Yaskawa INFORM job: A_ROOF_SIDE_0617_2_PAINT_4.JBI

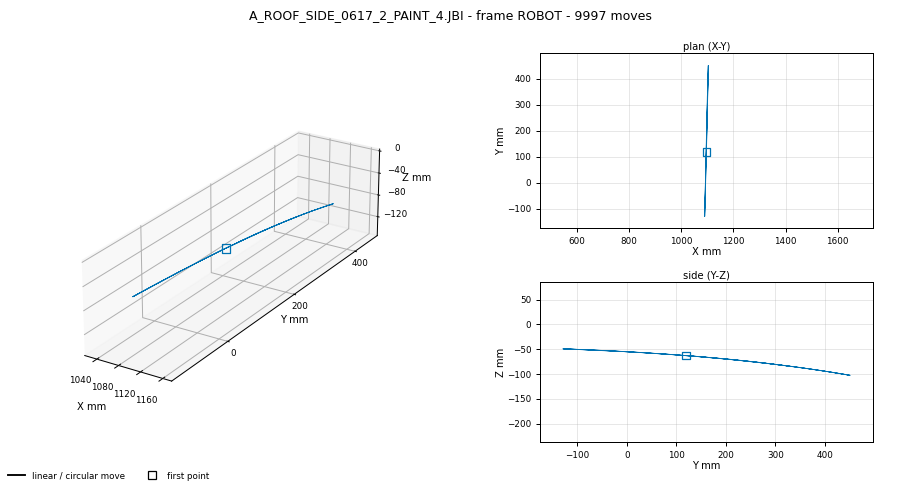
[picture p0: tool path of A_ROOF_SIDE_0617_2_PAINT_4.JBI in frame ROBOT, 9997 of 9997 moves have a stored position in this frame; points joined in program order, loops and branches not executed]
/JOB
//NAME A_ROOF_SIDE_0617_2_PAINT4
//POS
///NPOS 9997,0,0,0,0,0
///TOOL 1
///USER 0
///POSTYPE ROBOT
///RECTAN
///RCONF 1,0,0,0,0,0,0,0,0,0,0,0,0,0,0,0,0,0,0,0,0,0,0,0
C00000=1096.591,119.908,-62.578,176.519,16.757,152.269
C00001=1096.596,120.158,-62.598,176.522,16.758,152.268
C00002=1096.602,120.407,-62.618,176.524,16.758,152.268
C00003=1096.608,120.656,-62.637,176.527,16.758,152.267
C00004=1096.614,120.905,-62.656,176.530,16.759,152.267
C00005=1096.619,121.154,-62.675,176.533,16.759,152.267
C00006=1096.625,121.404,-62.694,176.536,16.760,152.266
C00007=1096.630,121.653,-62.713,176.539,16.761,152.266
C00008=1096.636,121.902,-62.733,176.541,16.761,152.265
C00009=1096.641,122.152,-62.753,176.544,16.762,152.265
C00010=1096.646,122.400,-62.772,176.546,16.761,152.264
C00011=1096.652,122.650,-62.791,176.549,16.762,152.264
C00012=1096.658,122.899,-62.811,176.552,16.763,152.263
C00013=1096.664,123.148,-62.830,176.555,16.763,152.263
C00014=1096.669,123.397,-62.850,176.558,16.764,152.262
C00015=1096.675,123.647,-62.869,176.561,16.764,152.262
C00016=1096.681,123.896,-62.889,176.563,16.765,152.262
C00017=1096.686,124.144,-62.908,176.566,16.765,152.261
C00018=1096.692,124.394,-62.927,176.569,16.766,152.261
C00019=1096.697,124.643,-62.946,176.571,16.766,152.260
C00020=1096.703,124.892,-62.966,176.575,16.766,152.260
C00021=1096.709,125.141,-62.985,176.578,16.767,152.259
C00022=1096.715,125.391,-63.005,176.580,16.767,152.259
C00023=1096.720,125.640,-63.025,176.583,16.768,152.258
C00024=1096.726,125.889,-63.045,176.585,16.768,152.258
C00025=1096.731,126.138,-63.064,176.589,16.768,152.257
C00026=1096.737,126.387,-63.083,176.592,16.769,152.257
C00027=1096.743,126.636,-63.103,176.594,16.769,152.256
C00028=1096.749,126.885,-63.123,176.597,16.770,152.256
C00029=1096.754,127.135,-63.142,176.600,16.770,152.256
C00030=1096.760,127.383,-63.162,176.602,16.770,152.255
C00031=1096.766,127.659,-63.183,176.606,16.771,152.254
C00032=1096.773,127.934,-63.205,176.609,16.771,152.254
C00033=1096.779,128.209,-63.226,176.612,16.772,152.253
C00034=1096.785,128.484,-63.249,176.615,16.772,152.253
C00035=1096.791,128.733,-63.269,176.618,16.773,152.252
C00036=1096.796,128.982,-63.288,176.621,16.773,152.252
C00037=1096.802,129.231,-63.307,176.624,16.773,152.251
C00038=1096.808,129.480,-63.327,176.627,16.774,152.251
C00039=1096.814,129.729,-63.347,176.629,16.774,152.250
C00040=1096.819,129.979,-63.366,176.632,16.774,152.250
C00041=1096.825,130.227,-63.386,176.636,16.775,152.249
C00042=1096.830,130.477,-63.406,176.638,16.775,152.249
C00043=1096.836,130.726,-63.426,176.641,16.775,152.248
C00044=1096.842,130.975,-63.445,176.644,16.776,152.248
C00045=1096.848,131.225,-63.465,176.646,16.776,152.247
C00046=1096.854,131.474,-63.486,176.649,16.777,152.247
C00047=1096.859,131.723,-63.505,176.653,16.777,152.246
C00048=1096.865,131.972,-63.525,176.655,16.777,152.246
C00049=1096.871,132.221,-63.544,176.658,16.778,152.245
C00050=1096.876,132.470,-63.565,176.661,16.778,152.245
C00051=1096.882,132.719,-63.585,176.664,16.778,152.244
C00052=1096.888,132.969,-63.604,176.667,16.778,152.244
C00053=1096.893,133.218,-63.624,176.670,16.779,152.243
C00054=1096.899,133.467,-63.644,176.672,16.779,152.243
C00055=1096.904,133.716,-63.664,176.676,16.779,152.242
C00056=1096.910,133.965,-63.684,176.679,16.780,152.242
C00057=1096.916,134.214,-63.704,176.681,16.780,152.241
C00058=1096.921,134.464,-63.724,176.684,16.781,152.241
C00059=1096.927,134.713,-63.744,176.687,16.781,152.240
C00060=1096.932,134.962,-63.765,176.690,16.781,152.240
C00061=1096.938,135.211,-63.784,176.693,16.782,152.239
C00062=1096.944,135.460,-63.804,176.696,16.782,152.239
C00063=1096.949,135.709,-63.824,176.698,16.782,152.238
C00064=1096.955,135.958,-63.844,176.701,16.783,152.238
C00065=1096.961,136.207,-63.865,176.705,16.783,152.237
C00066=1096.966,136.456,-63.884,176.707,16.783,152.237
C00067=1096.972,136.706,-63.905,176.710,16.784,152.236
C00068=1096.978,136.954,-63.925,176.713,16.784,152.236
C00069=1096.983,137.204,-63.945,176.716,16.785,152.235
C00070=1096.989,137.452,-63.965,176.719,16.785,152.235
C00071=1096.994,137.702,-63.984,176.722,16.785,152.234
C00072=1097.000,137.951,-64.005,176.725,16.785,152.234
C00073=1097.006,138.200,-64.025,176.727,16.785,152.233
C00074=1097.012,138.450,-64.046,176.731,16.786,152.233
C00075=1097.018,138.698,-64.066,176.734,16.786,152.232
C00076=1097.023,138.947,-64.086,176.736,16.786,152.232
C00077=1097.029,139.196,-64.106,176.739,16.787,152.231
C00078=1097.034,139.446,-64.126,176.743,16.787,152.231
C00079=1097.039,139.695,-64.147,176.745,16.787,152.230
C00080=1097.045,139.944,-64.167,176.748,16.788,152.230
C00081=1097.050,140.193,-64.187,176.751,16.788,152.229
C00082=1097.056,140.442,-64.207,176.755,16.788,152.228
C00083=1097.062,140.692,-64.228,176.757,16.788,152.228
C00084=1097.068,140.941,-64.248,176.760,16.789,152.227
C00085=1097.073,141.190,-64.269,176.763,16.789,152.227
C00086=1097.079,141.439,-64.289,176.766,16.789,152.226
C00087=1097.085,141.688,-64.309,176.769,16.790,152.226
C00088=1097.090,141.937,-64.330,176.772,16.790,152.225
C00089=1097.095,142.186,-64.350,176.775,16.790,152.225
C00090=1097.101,142.435,-64.370,176.778,16.790,152.224
C00091=1097.107,142.684,-64.391,176.781,16.791,152.224
C00092=1097.112,142.934,-64.412,176.784,16.791,152.223
C00093=1097.118,143.182,-64.432,176.786,16.791,152.223
C00094=1097.124,143.432,-64.452,176.790,16.792,152.222
C00095=1097.130,143.707,-64.475,176.793,16.792,152.222
C00096=1097.136,143.981,-64.497,176.797,16.792,152.221
C00097=1097.142,144.256,-64.520,176.800,16.792,152.220
C00098=1097.149,144.530,-64.542,176.803,16.793,152.220
C00099=1097.154,144.780,-64.563,176.806,16.793,152.219
C00100=1097.160,145.029,-64.584,176.809,16.793,152.219
C00101=1097.165,145.278,-64.604,176.812,16.793,152.218
C00102=1097.171,145.527,-64.624,176.815,16.794,152.218
C00103=1097.176,145.776,-64.645,176.817,16.794,152.217
C00104=1097.182,146.025,-64.667,176.821,16.794,152.216
C00105=1097.188,146.274,-64.686,176.824,16.795,152.216
C00106=1097.194,146.523,-64.707,176.827,16.795,152.215
C00107=1097.199,146.772,-64.728,176.830,16.795,152.215
C00108=1097.205,147.022,-64.749,176.833,16.795,152.214
C00109=1097.211,147.270,-64.769,176.836,16.795,152.214
C00110=1097.216,147.519,-64.790,176.839,16.795,152.213
C00111=1097.222,147.769,-64.810,176.842,16.796,152.213
C00112=1097.227,148.018,-64.831,176.845,16.796,152.212
C00113=1097.234,148.267,-64.852,176.848,16.796,152.211
C00114=1097.239,148.516,-64.872,176.851,16.796,152.211
C00115=1097.244,148.765,-64.893,176.854,16.796,152.210
C00116=1097.250,149.015,-64.914,176.857,16.797,152.210
C00117=1097.256,149.263,-64.935,176.861,16.797,152.209
C00118=1097.261,149.512,-64.956,176.863,16.797,152.209
C00119=1097.266,149.761,-64.976,176.866,16.797,152.208
C00120=1097.273,150.010,-64.997,176.870,16.798,152.207
C00121=1097.278,150.259,-65.018,176.872,16.797,152.207
C00122=1097.284,150.509,-65.038,176.875,16.798,152.206
C00123=1097.289,150.757,-65.060,176.879,16.798,152.206
C00124=1097.295,151.007,-65.081,176.882,16.799,152.205
C00125=1097.301,151.255,-65.102,176.884,16.798,152.205
C00126=1097.306,151.505,-65.122,176.888,16.799,152.204
C00127=1097.312,151.754,-65.143,176.891,16.799,152.203
C00128=1097.317,152.003,-65.165,176.894,16.799,152.203
C00129=1097.322,152.252,-65.185,176.897,16.799,152.202
C00130=1097.329,152.501,-65.207,176.900,16.800,152.202
C00131=1097.334,152.750,-65.227,176.903,16.800,152.201
C00132=1097.339,152.999,-65.249,176.906,16.800,152.201
C00133=1097.345,153.248,-65.269,176.909,16.800,152.200
C00134=1097.351,153.497,-65.290,176.912,16.801,152.200
C00135=1097.357,153.746,-65.311,176.915,16.801,152.199
C00136=1097.362,153.995,-65.331,176.918,16.800,152.198
C00137=1097.368,154.244,-65.353,176.921,16.801,152.198
C00138=1097.374,154.493,-65.374,176.925,16.801,152.197
C00139=1097.380,154.743,-65.395,176.928,16.801,152.197
C00140=1097.385,154.991,-65.416,176.930,16.801,152.196
C00141=1097.391,155.240,-65.437,176.934,16.801,152.195
C00142=1097.397,155.489,-65.459,176.937,16.802,152.195
C00143=1097.402,155.739,-65.479,176.940,16.802,152.194
C00144=1097.407,155.987,-65.501,176.943,16.802,152.194
C00145=1097.413,156.237,-65.522,176.946,16.802,152.193
C00146=1097.418,156.486,-65.543,176.949,16.802,152.192
C00147=1097.424,156.735,-65.565,176.953,16.803,152.192
C00148=1097.430,156.984,-65.585,176.955,16.802,152.191
C00149=1097.435,157.233,-65.607,176.958,16.803,152.191
C00150=1097.441,157.482,-65.628,176.962,16.803,152.190
C00151=1097.447,157.731,-65.649,176.965,16.803,152.190
C00152=1097.452,157.979,-65.670,176.968,16.803,152.189
C00153=1097.458,158.229,-65.692,176.971,16.803,152.188
C00154=1097.463,158.478,-65.713,176.974,16.804,152.188
C00155=1097.469,158.727,-65.735,176.978,16.804,152.187
C00156=1097.475,158.976,-65.756,176.980,16.803,152.187
C00157=1097.480,159.226,-65.777,176.983,16.804,152.186
C00158=1097.486,159.474,-65.798,176.987,16.804,152.185
C00159=1097.493,159.748,-65.822,176.990,16.804,152.185
C00160=1097.499,160.023,-65.845,176.994,16.804,152.184
C00161=1097.505,160.298,-65.868,176.997,16.804,152.183
C00162=1097.510,160.572,-65.893,177.001,16.804,152.183
C00163=1097.517,160.822,-65.914,177.004,16.805,152.182
C00164=1097.522,161.070,-65.936,177.007,16.805,152.181
C00165=1097.528,161.320,-65.956,177.010,16.804,152.181
C00166=1097.533,161.568,-65.978,177.013,16.805,152.180
C00167=1097.538,161.817,-66.000,177.016,16.805,152.180
C00168=1097.544,162.066,-66.021,177.020,16.805,152.179
C00169=1097.550,162.315,-66.042,177.023,16.805,152.178
C00170=1097.555,162.564,-66.065,177.026,16.805,152.178
C00171=1097.561,162.814,-66.085,177.029,16.806,152.177
C00172=1097.566,163.063,-66.107,177.032,16.806,152.177
C00173=1097.572,163.312,-66.129,177.036,16.806,152.176
C00174=1097.577,163.560,-66.150,177.038,16.806,152.175
C00175=1097.583,163.810,-66.172,177.041,16.806,152.175
C00176=1097.588,164.058,-66.194,177.045,16.806,152.174
C00177=1097.594,164.308,-66.216,177.048,16.806,152.174
C00178=1097.599,164.556,-66.237,177.051,16.807,152.173
C00179=1097.605,164.806,-66.259,177.054,16.807,152.173
C00180=1097.610,165.054,-66.281,177.057,16.807,152.172
C00181=1097.616,165.303,-66.302,177.061,16.807,152.171
C00182=1097.621,165.552,-66.324,177.064,16.807,152.171
C00183=1097.627,165.801,-66.346,177.067,16.808,152.170
C00184=1097.632,166.050,-66.368,177.070,16.807,152.169
C00185=1097.638,166.299,-66.389,177.073,16.807,152.169
C00186=1097.643,166.548,-66.411,177.076,16.808,152.168
C00187=1097.649,166.797,-66.433,177.080,16.808,152.168
C00188=1097.654,167.046,-66.455,177.083,16.808,152.167
C00189=1097.660,167.295,-66.476,177.086,16.807,152.166
C00190=1097.665,167.544,-66.498,177.089,16.808,152.166
C00191=1097.671,167.793,-66.520,177.093,16.808,152.165
C00192=1097.676,168.042,-66.542,177.096,16.808,152.164
C00193=1097.682,168.291,-66.563,177.099,16.809,152.164
C00194=1097.687,168.540,-66.585,177.102,16.808,152.163
C00195=1097.693,168.790,-66.607,177.105,16.808,152.163
C00196=1097.698,169.038,-66.629,177.109,16.809,152.162
C00197=1097.704,169.288,-66.650,177.112,16.809,152.161
C00198=1097.709,169.536,-66.673,177.115,16.808,152.161
C00199=1097.716,169.785,-66.694,177.118,16.808,152.160
C00200=1097.721,170.034,-66.717,177.121,16.809,152.159
C00201=1097.727,170.283,-66.738,177.125,16.809,152.159
C00202=1097.732,170.532,-66.760,177.128,16.809,152.158
C00203=1097.738,170.780,-66.782,177.131,16.808,152.158
C00204=1097.743,171.030,-66.804,177.134,16.809,152.157
C00205=1097.749,171.279,-66.827,177.138,16.809,152.156
C00206=1097.754,171.528,-66.848,177.141,16.809,152.156
C00207=1097.760,171.777,-66.871,177.144,16.809,152.155
C00208=1097.766,172.026,-66.892,177.148,16.809,152.154
C00209=1097.771,172.275,-66.914,177.150,16.809,152.154
C00210=1097.777,172.524,-66.936,177.154,16.809,152.153
C00211=1097.782,172.772,-66.958,177.157,16.809,152.152
C00212=1097.788,173.022,-66.981,177.161,16.810,152.152
C00213=1097.794,173.271,-67.002,177.164,16.809,152.151
C00214=1097.799,173.519,-67.025,177.167,16.809,152.150
C00215=1097.805,173.768,-67.047,177.170,16.809,152.150
C00216=1097.811,174.018,-67.069,177.174,16.809,152.149
C00217=1097.816,174.267,-67.092,177.177,16.810,152.149
C00218=1097.822,174.515,-67.113,177.180,16.809,152.148
C00219=1097.827,174.765,-67.135,177.183,16.809,152.147
C00220=1097.833,175.014,-67.158,177.186,16.809,152.147
C00221=1097.839,175.262,-67.179,177.190,16.809,152.146
C00222=1097.844,175.511,-67.202,177.193,16.809,152.145
C00223=1097.851,175.785,-67.226,177.197,16.809,152.144
C00224=1097.857,176.060,-67.251,177.201,16.809,152.144
C00225=1097.864,176.334,-67.276,177.204,16.809,152.143
C00226=1097.869,176.608,-67.300,177.208,16.809,152.142
C00227=1097.875,176.857,-67.323,177.211,16.809,152.142
C00228=1097.881,177.106,-67.344,177.214,16.809,152.141
C00229=1097.887,177.355,-67.367,177.218,16.809,152.140
C00230=1097.892,177.604,-67.389,177.222,16.809,152.140
C00231=1097.898,177.852,-67.411,177.224,16.809,152.139
C00232=1097.903,178.102,-67.434,177.228,16.809,152.138
C00233=1097.909,178.351,-67.457,177.231,16.809,152.138
C00234=1097.914,178.600,-67.479,177.234,16.809,152.137
C00235=1097.920,178.848,-67.501,177.238,16.809,152.136
C00236=1097.926,179.097,-67.524,177.241,16.809,152.136
C00237=1097.931,179.346,-67.546,177.244,16.808,152.135
C00238=1097.938,179.595,-67.568,177.248,16.808,152.134
C00239=1097.943,179.845,-67.591,177.251,16.809,152.134
C00240=1097.949,180.093,-67.614,177.254,16.809,152.133
C00241=1097.954,180.342,-67.636,177.258,16.809,152.132
C00242=1097.960,180.591,-67.658,177.262,16.809,152.131
C00243=1097.966,180.840,-67.681,177.264,16.808,152.131
C00244=1097.972,181.089,-67.704,177.268,16.808,152.130
C00245=1097.977,181.338,-67.726,177.271,16.808,152.129
C00246=1097.984,181.587,-67.748,177.275,16.808,152.129
C00247=1097.989,181.836,-67.771,177.278,16.808,152.128
C00248=1097.994,182.084,-67.793,177.282,16.808,152.127
C00249=1098.000,182.333,-67.816,177.284,16.808,152.127
C00250=1098.006,182.582,-67.838,177.288,16.808,152.126
C00251=1098.012,182.831,-67.861,177.291,16.808,152.125
C00252=1098.018,183.080,-67.883,177.295,16.808,152.125
C00253=1098.023,183.329,-67.906,177.298,16.808,152.124
C00254=1098.029,183.578,-67.929,177.302,16.808,152.123
C00255=1098.036,183.827,-67.952,177.305,16.807,152.123
C00256=1098.041,184.076,-67.975,177.308,16.807,152.122
C00257=1098.047,184.325,-67.997,177.312,16.807,152.121
C00258=1098.052,184.573,-68.019,177.315,16.807,152.120
C00259=1098.058,184.822,-68.042,177.319,16.807,152.120
C00260=1098.063,185.071,-68.065,177.322,16.807,152.119
C00261=1098.069,185.320,-68.088,177.325,16.806,152.118
C00262=1098.075,185.569,-68.111,177.328,16.807,152.118
C00263=1098.080,185.818,-68.134,177.332,16.807,152.117
C00264=1098.086,186.067,-68.156,177.335,16.807,152.116
C00265=1098.092,186.316,-68.179,177.339,16.807,152.116
C00266=1098.097,186.564,-68.202,177.342,16.807,152.115
C00267=1098.102,186.813,-68.225,177.346,16.807,152.114
C00268=1098.108,187.062,-68.248,177.349,16.807,152.114
C00269=1098.113,187.311,-68.271,177.352,16.806,152.113
C00270=1098.119,187.560,-68.294,177.355,16.806,152.112
C00271=1098.125,187.809,-68.317,177.359,16.806,152.111
C00272=1098.130,188.058,-68.340,177.362,16.807,152.111
C00273=1098.136,188.306,-68.363,177.366,16.807,152.110
C00274=1098.141,188.555,-68.386,177.369,16.807,152.109
C00275=1098.147,188.804,-68.409,177.373,16.807,152.109
C00276=1098.152,189.053,-68.432,177.376,16.806,152.108
C00277=1098.158,189.302,-68.455,177.379,16.806,152.107
C00278=1098.163,189.551,-68.478,177.383,16.806,152.107
C00279=1098.169,189.800,-68.501,177.386,16.806,152.106
C00280=1098.175,190.049,-68.524,177.389,16.806,152.105
C00281=1098.180,190.298,-68.548,177.393,16.806,152.105
C00282=1098.186,190.547,-68.571,177.397,16.806,152.104
C00283=1098.191,190.796,-68.593,177.400,16.806,152.103
C00284=1098.197,191.045,-68.616,177.404,16.806,152.102
C00285=1098.203,191.294,-68.639,177.406,16.805,152.102
C00286=1098.208,191.542,-68.664,177.410,16.805,152.101
C00287=1098.214,191.816,-68.689,177.413,16.805,152.100
C00288=1098.220,192.090,-68.714,177.418,16.805,152.099
C00289=1098.226,192.363,-68.740,177.422,16.805,152.099
C00290=1098.232,192.637,-68.765,177.425,16.805,152.098
C00291=1098.238,192.886,-68.788,177.429,16.805,152.097
C00292=1098.243,193.135,-68.811,177.433,16.805,152.096
C00293=1098.249,193.384,-68.834,177.436,16.805,152.096
C00294=1098.255,193.632,-68.858,177.440,16.805,152.095
C00295=1098.261,193.881,-68.881,177.442,16.804,152.094
C00296=1098.266,194.130,-68.905,177.446,16.804,152.094
C00297=1098.271,194.379,-68.928,177.449,16.804,152.093
C00298=1098.277,194.628,-68.951,177.453,16.804,152.092
C00299=1098.283,194.877,-68.974,177.456,16.804,152.091
C00300=1098.289,195.126,-68.998,177.460,16.804,152.091
C00301=1098.295,195.375,-69.022,177.464,16.804,152.090
C00302=1098.301,195.624,-69.045,177.467,16.804,152.089
C00303=1098.306,195.873,-69.068,177.471,16.804,152.089
C00304=1098.312,196.121,-69.092,177.473,16.803,152.088
C00305=1098.317,196.370,-69.115,177.477,16.803,152.087
C00306=1098.322,196.619,-69.138,177.480,16.803,152.087
C00307=1098.328,196.867,-69.162,177.484,16.803,152.086
C00308=1098.334,197.116,-69.185,177.487,16.803,152.085
C00309=1098.339,197.366,-69.208,177.491,16.803,152.084
C00310=1098.345,197.614,-69.232,177.495,16.803,152.083
C00311=1098.351,197.863,-69.255,177.498,16.803,152.083
C00312=1098.357,198.112,-69.280,177.502,16.803,152.082
C00313=1098.362,198.361,-69.303,177.505,16.803,152.081
C00314=1098.368,198.609,-69.326,177.508,16.802,152.081
C00315=1098.373,198.858,-69.350,177.512,16.802,152.080
C00316=1098.380,199.107,-69.374,177.516,16.802,152.079
C00317=1098.384,199.356,-69.397,177.519,16.802,152.078
C00318=1098.391,199.605,-69.421,177.523,16.802,152.078
C00319=1098.397,199.854,-69.444,177.526,16.802,152.077
C00320=1098.402,200.102,-69.468,177.530,16.802,152.076
C00321=1098.408,200.351,-69.491,177.533,16.801,152.075
C00322=1098.414,200.600,-69.515,177.537,16.801,152.075
C00323=1098.419,200.849,-69.538,177.541,16.801,152.074
C00324=1098.426,201.098,-69.562,177.544,16.801,152.073
C00325=1098.431,201.347,-69.586,177.547,16.800,152.072
C00326=1098.437,201.595,-69.610,177.551,16.800,152.072
C00327=1098.442,201.844,-69.634,177.554,16.800,152.071
C00328=1098.448,202.093,-69.657,177.558,16.800,152.070
C00329=1098.454,202.342,-69.681,177.562,16.800,152.069
C00330=1098.460,202.590,-69.705,177.565,16.800,152.069
C00331=1098.465,202.839,-69.728,177.569,16.799,152.068
C00332=1098.471,203.088,-69.752,177.572,16.799,152.067
C00333=1098.476,203.337,-69.777,177.576,16.799,152.067
C00334=1098.482,203.586,-69.800,177.580,16.799,152.066
C00335=1098.488,203.835,-69.824,177.583,16.799,152.065
C00336=1098.494,204.083,-69.848,177.587,16.799,152.064
C00337=1098.499,204.332,-69.871,177.590,16.799,152.064
C00338=1098.504,204.581,-69.896,177.594,16.799,152.063
C00339=1098.510,204.830,-69.920,177.597,16.798,152.062
C00340=1098.516,205.078,-69.944,177.600,16.798,152.061
C00341=1098.521,205.327,-69.967,177.604,16.798,152.061
C00342=1098.527,205.576,-69.991,177.607,16.798,152.060
C00343=1098.533,205.825,-70.016,177.611,16.797,152.059
C00344=1098.538,206.074,-70.040,177.615,16.797,152.058
C00345=1098.544,206.322,-70.063,177.618,16.797,152.058
C00346=1098.549,206.571,-70.087,177.622,16.797,152.057
C00347=1098.555,206.820,-70.112,177.626,16.797,152.056
C00348=1098.561,207.069,-70.135,177.629,16.797,152.055
C00349=1098.566,207.317,-70.160,177.633,16.797,152.055
C00350=1098.572,207.566,-70.184,177.636,16.797,152.054
C00351=1098.595,208.576,-70.282,177.680,16.812,152.049
C00352=1098.603,208.947,-70.318,177.685,16.813,152.048
C00353=1098.611,209.317,-70.354,177.690,16.814,152.047
C00354=1098.620,209.688,-70.390,177.695,16.815,152.046
C00355=1098.629,210.058,-70.427,177.699,16.816,152.045
C00356=1098.634,210.306,-70.451,177.703,16.817,152.045
C00357=1098.640,210.555,-70.476,177.707,16.817,152.044
C00358=1098.645,210.804,-70.500,177.710,16.818,152.044
C00359=1098.651,211.053,-70.524,177.713,16.818,152.043
C00360=1098.657,211.302,-70.549,177.717,16.820,152.043
C00361=1098.662,211.550,-70.573,177.720,16.820,152.042
C00362=1098.668,211.799,-70.599,177.723,16.821,152.042
C00363=1098.673,212.048,-70.623,177.726,16.821,152.041
C00364=1098.679,212.296,-70.647,177.730,16.822,152.041
C00365=1098.685,212.546,-70.672,177.734,16.823,152.040
C00366=1098.690,212.794,-70.696,177.737,16.824,152.040
C00367=1098.696,213.043,-70.721,177.740,16.824,152.039
C00368=1098.701,213.291,-70.746,177.744,16.825,152.039
C00369=1098.707,213.541,-70.770,177.747,16.826,152.038
C00370=1098.713,213.789,-70.795,177.750,16.826,152.038
C00371=1098.718,214.037,-70.820,177.753,16.827,152.037
C00372=1098.724,214.287,-70.844,177.757,16.828,152.037
C00373=1098.729,214.535,-70.868,177.761,16.829,152.036
C00374=1098.736,214.784,-70.894,177.764,16.830,152.036
C00375=1098.741,215.032,-70.918,177.768,16.831,152.035
C00376=1098.747,215.282,-70.943,177.771,16.831,152.034
C00377=1098.752,215.530,-70.968,177.774,16.832,152.034
C00378=1098.757,215.779,-70.992,177.777,16.832,152.034
C00379=1098.763,216.028,-71.017,177.781,16.834,152.033
C00380=1098.768,216.276,-71.042,177.784,16.834,152.032
C00381=1098.774,216.525,-71.067,177.787,16.835,152.032
C00382=1098.780,216.773,-71.092,177.790,16.835,152.032
C00383=1098.786,217.022,-71.116,177.794,16.836,152.031
C00384=1098.791,217.271,-71.142,177.798,16.837,152.030
C00385=1098.797,217.520,-71.166,177.801,16.838,152.030
C00386=1098.802,217.768,-71.191,177.805,16.839,152.029
C00387=1098.808,218.017,-71.216,177.808,16.839,152.029
C00388=1098.814,218.265,-71.241,177.811,16.840,152.028
C00389=1098.819,218.515,-71.266,177.815,16.841,152.028
C00390=1098.825,218.763,-71.292,177.818,16.842,152.027
C00391=1098.830,219.012,-71.316,177.821,16.842,152.027
C00392=1098.837,219.261,-71.341,177.825,16.843,152.026
C00393=1098.842,219.509,-71.365,177.828,16.844,152.026
C00394=1098.847,219.758,-71.391,177.832,16.845,152.025
C00395=1098.853,220.007,-71.416,177.835,16.845,152.025
C00396=1098.859,220.256,-71.441,177.839,16.846,152.024
C00397=1098.865,220.504,-71.466,177.842,16.847,152.024
C00398=1098.870,220.753,-71.491,177.845,16.848,152.023
C00399=1098.876,221.002,-71.516,177.848,16.848,152.023
C00400=1098.881,221.250,-71.541,177.852,16.849,152.022
C00401=1098.887,221.499,-71.566,177.856,16.850,152.022
C00402=1098.893,221.748,-71.592,177.858,16.851,152.021
C00403=1098.898,221.996,-71.617,177.863,16.852,152.021
C00404=1098.907,222.371,-71.654,177.868,16.853,152.020
C00405=1098.915,222.745,-71.692,177.873,16.854,152.019
C00406=1098.923,223.119,-71.731,177.878,16.855,152.018
C00407=1098.932,223.494,-71.769,177.883,16.857,152.018
C00408=1098.937,223.742,-71.794,177.886,16.857,152.017
C00409=1098.943,223.991,-71.819,177.889,16.857,152.017
C00410=1098.949,224.240,-71.844,177.893,16.859,152.016
C00411=1098.954,224.488,-71.870,177.896,16.859,152.016
C00412=1098.960,224.737,-71.895,177.900,16.860,152.015
C00413=1098.966,224.986,-71.921,177.903,16.861,152.015
C00414=1098.971,225.234,-71.946,177.907,16.862,152.014
C00415=1098.977,225.484,-71.971,177.910,16.862,152.014
C00416=1098.982,225.731,-71.996,177.914,16.864,152.013
C00417=1098.988,225.980,-72.022,177.917,16.864,152.013
C00418=1098.994,226.229,-72.047,177.920,16.865,152.012
C00419=1098.999,226.478,-72.073,177.924,16.866,152.012
C00420=1099.005,226.726,-72.098,177.927,16.867,152.011
C00421=1099.010,226.975,-72.124,177.930,16.867,152.011
C00422=1099.017,227.224,-72.150,177.934,16.869,152.010
C00423=1099.022,227.472,-72.175,177.937,16.869,152.010
C00424=1099.028,227.721,-72.200,177.940,16.870,152.009
C00425=1099.033,227.970,-72.226,177.944,16.871,152.009
C00426=1099.039,228.218,-72.252,177.947,16.872,152.008
C00427=1099.044,228.467,-72.277,177.951,16.873,152.008
C00428=1099.051,228.715,-72.303,177.955,16.873,152.007
C00429=1099.056,228.964,-72.329,177.958,16.874,152.007
C00430=1099.062,229.213,-72.354,177.962,16.875,152.006
C00431=1099.067,229.461,-72.379,177.965,16.876,152.006
C00432=1099.073,229.710,-72.405,177.968,16.876,152.005
C00433=1099.079,229.959,-72.431,177.972,16.878,152.005
C00434=1099.084,230.208,-72.457,177.975,16.878,152.004
C00435=1099.090,230.456,-72.482,177.978,16.879,152.004
C00436=1099.095,230.705,-72.508,177.982,16.880,152.003
C00437=1099.101,230.954,-72.533,177.985,16.881,152.003
C00438=1099.107,231.202,-72.560,177.989,16.882,152.002
C00439=1099.112,231.450,-72.585,177.992,16.883,152.002
C00440=1099.118,231.699,-72.611,177.995,16.883,152.001
C00441=1099.124,231.948,-72.636,177.999,16.885,152.001
C00442=1099.129,232.197,-72.662,178.002,16.885,152.000
C00443=1099.135,232.445,-72.689,178.006,16.886,152.000
C00444=1099.141,232.693,-72.714,178.009,16.887,151.999
C00445=1099.146,232.942,-72.740,178.013,16.888,151.999
C00446=1099.152,233.191,-72.766,178.017,16.889,151.998
C00447=1099.157,233.440,-72.792,178.020,16.890,151.998
C00448=1099.164,233.688,-72.818,178.023,16.890,151.997
C00449=1099.168,233.936,-72.843,178.027,16.891,151.997
C00450=1099.174,234.185,-72.869,178.030,16.892,151.996
C00451=1099.180,234.434,-72.896,178.034,16.893,151.996
C00452=1099.185,234.683,-72.922,178.037,16.894,151.995
C00453=1099.191,234.931,-72.947,178.040,16.895,151.995
C00454=1099.197,235.180,-72.974,178.044,16.896,151.994
C00455=1099.202,235.428,-72.999,178.047,16.897,151.994
C00456=1099.211,235.794,-73.038,178.052,16.898,151.993
C00457=1099.218,236.160,-73.077,178.057,16.899,151.992
C00458=1099.227,236.526,-73.115,178.062,16.901,151.992
C00459=1099.235,236.891,-73.153,178.067,16.902,151.991
C00460=1099.241,237.140,-73.179,178.071,16.903,151.991
C00461=1099.246,237.389,-73.206,178.074,16.904,151.990
C00462=1099.252,237.638,-73.232,178.077,16.905,151.990
C00463=1099.258,237.886,-73.258,178.081,16.906,151.989
C00464=1099.263,238.134,-73.284,178.084,16.907,151.989
C00465=1099.269,238.382,-73.310,178.088,16.908,151.988
C00466=1099.275,238.631,-73.336,178.091,16.909,151.988
C00467=1099.280,238.880,-73.363,178.094,16.909,151.987
C00468=1099.286,239.129,-73.389,178.098,16.911,151.987
C00469=1099.292,239.377,-73.415,178.101,16.911,151.986
C00470=1099.297,239.626,-73.441,178.105,16.913,151.986
C00471=1099.303,239.874,-73.468,178.109,16.913,151.985
C00472=1099.309,240.123,-73.494,178.112,16.915,151.985
C00473=1099.314,240.372,-73.520,178.116,16.915,151.984
C00474=1099.320,240.620,-73.547,178.119,16.916,151.984
C00475=1099.325,240.869,-73.573,178.123,16.917,151.983
C00476=1099.331,241.118,-73.600,178.126,16.918,151.983
C00477=1099.337,241.366,-73.626,178.130,16.919,151.982
C00478=1099.342,241.615,-73.652,178.133,16.920,151.982
C00479=1099.348,241.863,-73.679,178.136,16.921,151.982
C00480=1099.354,242.112,-73.705,178.140,16.922,151.981
C00481=1099.360,242.360,-73.732,178.143,16.923,151.981
C00482=1099.365,242.609,-73.758,178.147,16.924,151.980
C00483=1099.371,242.857,-73.785,178.150,16.924,151.980
C00484=1099.377,243.106,-73.811,178.154,16.926,151.979
C00485=1099.382,243.354,-73.838,178.157,16.926,151.979
C00486=1099.387,243.603,-73.865,178.161,16.928,151.978
C00487=1099.393,243.852,-73.891,178.164,16.928,151.978
C00488=1099.399,244.100,-73.918,178.168,16.930,151.977
C00489=1099.405,244.348,-73.944,178.171,16.930,151.977
C00490=1099.410,244.597,-73.971,178.175,16.932,151.976
C00491=1099.416,244.846,-73.997,178.178,16.932,151.976
C00492=1099.421,245.094,-74.024,178.181,16.934,151.975
C00493=1099.427,245.343,-74.051,178.185,16.934,151.975
C00494=1099.432,245.591,-74.078,178.188,16.935,151.975
C00495=1099.438,245.839,-74.104,178.192,16.937,151.974
C00496=1099.444,246.088,-74.131,178.195,16.937,151.974
C00497=1099.449,246.336,-74.158,178.199,16.939,151.973
C00498=1099.455,246.585,-74.185,178.202,16.939,151.973
C00499=1099.460,246.833,-74.211,178.206,16.941,151.972
C00500=1099.466,247.082,-74.238,178.209,16.942,151.972
C00501=1099.472,247.331,-74.266,178.213,16.943,151.971
C00502=1099.478,247.579,-74.292,178.215,16.944,151.971
C00503=1099.483,247.828,-74.319,178.219,16.945,151.970
C00504=1099.488,248.076,-74.346,178.222,16.946,151.970
C00505=1099.494,248.325,-74.373,178.226,16.947,151.970
C00506=1099.499,248.573,-74.400,178.229,16.948,151.969
C00507=1099.505,248.822,-74.427,178.233,16.949,151.969
C00508=1099.513,249.180,-74.465,178.238,16.951,151.968
C00509=1099.521,249.540,-74.504,178.243,16.952,151.967
C00510=1099.529,249.899,-74.544,178.248,16.954,151.967
C00511=1099.537,250.257,-74.582,178.253,16.955,151.966
C00512=1099.542,250.506,-74.609,178.256,16.956,151.966
C00513=1099.548,250.754,-74.636,178.260,16.957,151.965
C00514=1099.553,251.003,-74.664,178.263,16.958,151.965
C00515=1099.560,251.252,-74.691,178.267,16.960,151.964
C00516=1099.565,251.500,-74.718,178.270,16.960,151.964
C00517=1099.570,251.749,-74.745,178.273,16.962,151.963
C00518=1099.576,251.997,-74.771,178.277,16.962,151.963
C00519=1099.582,252.245,-74.799,178.280,16.964,151.963
C00520=1099.587,252.493,-74.826,178.284,16.965,151.962
C00521=1099.593,252.743,-74.854,178.287,16.966,151.962
C00522=1099.599,252.991,-74.880,178.291,16.968,151.961
C00523=1099.604,253.239,-74.908,178.294,16.968,151.961
C00524=1099.610,253.488,-74.935,178.298,16.970,151.960
C00525=1099.615,253.736,-74.962,178.301,16.971,151.960
C00526=1099.621,253.985,-74.989,178.305,16.972,151.959
C00527=1099.627,254.233,-75.017,178.308,16.973,151.959
C00528=1099.632,254.482,-75.044,178.312,16.974,151.959
C00529=1099.638,254.730,-75.072,178.315,16.975,151.958
C00530=1099.643,254.978,-75.098,178.319,16.976,151.958
C00531=1099.649,255.227,-75.126,178.322,16.977,151.957
C00532=1099.654,255.476,-75.154,178.326,16.978,151.957
C00533=1099.660,255.724,-75.181,178.329,16.979,151.956
C00534=1099.666,255.972,-75.209,178.333,16.980,151.956
C00535=1099.672,256.221,-75.236,178.335,16.981,151.955
C00536=1099.677,256.470,-75.263,178.339,16.982,151.955
C00537=1099.683,256.717,-75.290,178.342,16.983,151.955
C00538=1099.688,256.966,-75.317,178.346,16.985,151.954
C00539=1099.694,257.215,-75.346,178.350,16.986,151.954
C00540=1099.700,257.463,-75.372,178.353,16.987,151.953
C00541=1099.705,257.711,-75.400,178.357,16.989,151.953
C00542=1099.712,257.960,-75.427,178.360,16.989,151.952
C00543=1099.717,258.208,-75.455,178.364,16.991,151.952
C00544=1099.722,258.456,-75.483,178.367,16.991,151.951
C00545=1099.729,258.705,-75.510,178.371,16.993,151.951
C00546=1099.734,258.954,-75.538,178.374,16.994,151.951
C00547=1099.740,259.202,-75.565,178.378,16.995,151.950
C00548=1099.746,259.451,-75.593,178.381,16.996,151.950
C00549=1099.751,259.699,-75.621,178.384,16.997,151.949
C00550=1099.757,259.947,-75.648,178.388,16.998,151.949
C00551=1099.763,260.196,-75.676,178.391,16.999,151.948
C00552=1099.768,260.444,-75.704,178.395,17.001,151.948
C00553=1099.774,260.692,-75.731,178.398,17.001,151.948
C00554=1099.780,260.941,-75.759,178.402,17.003,151.947
C00555=1099.785,261.189,-75.787,178.405,17.004,151.947
C00556=1099.791,261.438,-75.814,178.409,17.005,151.946
C00557=1099.797,261.686,-75.842,178.412,17.006,151.946
C00558=1099.802,261.934,-75.870,178.416,17.007,151.945
C00559=1099.808,262.183,-75.898,178.420,17.009,151.945
C00560=1099.816,262.539,-75.938,178.425,17.010,151.944
C00561=1099.825,262.895,-75.978,178.429,17.012,151.944
C00562=1099.833,263.251,-76.018,178.434,17.014,151.943
C00563=1099.841,263.607,-76.057,178.439,17.015,151.942
C00564=1099.846,263.856,-76.085,178.443,17.016,151.942
C00565=1099.853,264.104,-76.113,178.446,17.017,151.942
C00566=1099.858,264.352,-76.141,178.450,17.018,151.941
C00567=1099.864,264.601,-76.169,178.453,17.019,151.941
C00568=1099.870,264.849,-76.197,178.457,17.021,151.940
C00569=1099.875,265.097,-76.225,178.460,17.022,151.940
C00570=1099.881,265.346,-76.253,178.464,17.023,151.940
C00571=1099.886,265.594,-76.281,178.467,17.025,151.939
C00572=1099.892,265.842,-76.310,178.470,17.026,151.939
C00573=1099.897,266.091,-76.337,178.474,17.027,151.938
C00574=1099.904,266.340,-76.365,178.477,17.028,151.938
C00575=1099.909,266.588,-76.393,178.481,17.029,151.937
C00576=1099.915,266.836,-76.421,178.485,17.031,151.937
C00577=1099.921,267.084,-76.449,178.488,17.032,151.937
C00578=1099.926,267.332,-76.478,178.491,17.033,151.936
C00579=1099.932,267.581,-76.506,178.495,17.035,151.936
C00580=1099.938,267.829,-76.534,178.498,17.036,151.936
C00581=1099.944,268.077,-76.562,178.502,17.037,151.935
C00582=1099.949,268.325,-76.590,178.505,17.038,151.935
C00583=1099.955,268.574,-76.619,178.509,17.040,151.934
C00584=1099.960,268.822,-76.647,178.512,17.041,151.934
C00585=1099.966,269.071,-76.675,178.515,17.042,151.934
C00586=1099.971,269.319,-76.703,178.519,17.043,151.933
C00587=1099.977,269.567,-76.732,178.522,17.044,151.933
C00588=1099.982,269.816,-76.760,178.526,17.046,151.932
C00589=1099.988,270.064,-76.789,178.530,17.047,151.932
C00590=1099.994,270.312,-76.817,178.533,17.048,151.932
C00591=1099.999,270.561,-76.845,178.536,17.050,151.931
C00592=1100.006,270.809,-76.874,178.540,17.051,151.931
C00593=1100.011,271.057,-76.902,178.543,17.052,151.930
C00594=1100.017,271.306,-76.930,178.547,17.054,151.930
C00595=1100.022,271.554,-76.958,178.550,17.055,151.930
C00596=1100.028,271.803,-76.988,178.554,17.056,151.929
C00597=1100.033,272.051,-77.016,178.557,17.058,151.929
C00598=1100.039,272.299,-77.044,178.560,17.059,151.928
C00599=1100.045,272.547,-77.073,178.564,17.060,151.928
C00600=1100.051,272.795,-77.101,178.568,17.062,151.928
C00601=1100.057,273.044,-77.130,178.571,17.063,151.927
C00602=1100.062,273.292,-77.159,178.574,17.064,151.927
C00603=1100.068,273.541,-77.187,178.578,17.066,151.927
C00604=1100.073,273.789,-77.215,178.581,17.067,151.926
C00605=1100.079,274.037,-77.244,178.585,17.068,151.926
C00606=1100.084,274.286,-77.273,178.588,17.070,151.925
C00607=1100.090,274.533,-77.302,178.591,17.071,151.925
C00608=1100.096,274.782,-77.330,178.595,17.073,151.925
C00609=1100.102,275.030,-77.359,178.599,17.074,151.924
C00610=1100.107,275.279,-77.388,178.602,17.075,151.924
C00611=1100.113,275.527,-77.416,178.605,17.077,151.924
C00612=1100.121,275.885,-77.458,178.610,17.078,151.923
C00613=1100.129,276.245,-77.500,178.615,17.080,151.923
C00614=1100.137,276.603,-77.541,178.621,17.083,151.922
C00615=1100.145,276.962,-77.583,178.625,17.084,151.921
C00616=1100.151,277.210,-77.611,178.629,17.086,151.921
C00617=1100.156,277.459,-77.640,178.632,17.087,151.921
C00618=1100.163,277.707,-77.669,178.636,17.088,151.920
C00619=1100.168,277.955,-77.697,178.640,17.090,151.920
C00620=1100.173,278.203,-77.727,178.642,17.091,151.920
C00621=1100.180,278.451,-77.756,178.646,17.093,151.919
C00622=1100.184,278.700,-77.784,178.650,17.094,151.919
C00623=1100.191,278.948,-77.814,178.654,17.096,151.918
C00624=1100.196,279.196,-77.843,178.656,17.097,151.918
C00625=1100.201,279.444,-77.871,178.660,17.099,151.918
C00626=1100.208,279.693,-77.900,178.664,17.100,151.918
C00627=1100.213,279.941,-77.930,178.667,17.101,151.917
C00628=1100.219,280.190,-77.958,178.670,17.103,151.917
C00629=1100.224,280.438,-77.987,178.674,17.104,151.916
C00630=1100.230,280.686,-78.016,178.677,17.105,151.916
C00631=1100.236,280.934,-78.046,178.681,17.107,151.916
C00632=1100.241,281.182,-78.075,178.684,17.109,151.915
C00633=1100.247,281.431,-78.104,178.687,17.110,151.915
C00634=1100.253,281.679,-78.133,178.691,17.111,151.915
C00635=1100.258,281.927,-78.162,178.694,17.113,151.914
C00636=1100.264,282.175,-78.191,178.698,17.115,151.914
C00637=1100.270,282.423,-78.221,178.701,17.116,151.914
C00638=1100.275,282.671,-78.250,178.705,17.117,151.913
C00639=1100.281,282.920,-78.279,178.708,17.119,151.913
C00640=1100.286,283.168,-78.308,178.711,17.120,151.913
C00641=1100.292,283.416,-78.337,178.715,17.122,151.912
C00642=1100.298,283.665,-78.367,178.719,17.123,151.912
C00643=1100.303,283.913,-78.396,178.722,17.125,151.912
C00644=1100.309,284.160,-78.425,178.725,17.126,151.911
C00645=1100.314,284.409,-78.454,178.729,17.128,151.911
C00646=1100.320,284.657,-78.484,178.732,17.130,151.911
C00647=1100.326,284.905,-78.513,178.736,17.131,151.910
C00648=1100.332,285.154,-78.543,178.739,17.133,151.910
C00649=1100.337,285.402,-78.572,178.743,17.134,151.910
C00650=1100.343,285.650,-78.601,178.746,17.136,151.909
C00651=1100.348,285.898,-78.631,178.749,17.137,151.909
C00652=1100.354,286.147,-78.660,178.753,17.139,151.909
C00653=1100.360,286.394,-78.690,178.756,17.140,151.908
C00654=1100.365,286.642,-78.719,178.760,17.142,151.908
C00655=1100.371,286.890,-78.749,178.763,17.143,151.908
C00656=1100.377,287.138,-78.778,178.766,17.145,151.907
C00657=1100.383,287.387,-78.808,178.770,17.147,151.907
C00658=1100.388,287.635,-78.837,178.774,17.148,151.907
C00659=1100.394,287.884,-78.867,178.777,17.149,151.906
C00660=1100.400,288.131,-78.897,178.780,17.151,151.906
C00661=1100.405,288.379,-78.926,178.784,17.153,151.906
C00662=1100.411,288.627,-78.956,178.788,17.154,151.905
C00663=1100.416,288.876,-78.985,178.790,17.156,151.905
C00664=1100.425,289.245,-79.029,178.796,17.158,151.905
C00665=1100.433,289.613,-79.073,178.801,17.161,151.904
C00666=1100.442,289.981,-79.117,178.806,17.163,151.904
C00667=1100.450,290.348,-79.162,178.811,17.166,151.903
C00668=1100.456,290.596,-79.191,178.815,17.167,151.903
C00669=1100.462,290.845,-79.221,178.818,17.168,151.903
C00670=1100.467,291.093,-79.251,178.821,17.170,151.902
C00671=1100.473,291.341,-79.281,178.825,17.172,151.902
C00672=1100.478,291.590,-79.310,178.828,17.174,151.902
C00673=1100.484,291.837,-79.341,178.832,17.175,151.902
C00674=1100.490,292.086,-79.370,178.835,17.177,151.901
C00675=1100.496,292.334,-79.401,178.838,17.178,151.901
C00676=1100.501,292.582,-79.430,178.842,17.180,151.901
C00677=1100.507,292.831,-79.460,178.846,17.182,151.900
C00678=1100.512,293.078,-79.490,178.849,17.183,151.900
C00679=1100.518,293.327,-79.520,178.852,17.185,151.900
C00680=1100.523,293.574,-79.550,178.856,17.187,151.899
C00681=1100.529,293.822,-79.579,178.859,17.189,151.899
C00682=1100.535,294.070,-79.609,178.863,17.190,151.899
C00683=1100.541,294.318,-79.639,178.865,17.192,151.899
C00684=1100.547,294.566,-79.669,178.869,17.193,151.898
C00685=1100.552,294.814,-79.700,178.873,17.195,151.898
C00686=1100.557,295.063,-79.730,178.876,17.197,151.898
C00687=1100.563,295.310,-79.760,178.880,17.199,151.898
C00688=1100.569,295.559,-79.790,178.883,17.200,151.897
C00689=1100.574,295.807,-79.820,178.886,17.202,151.897
C00690=1100.580,296.055,-79.851,178.890,17.203,151.897
C00691=1100.586,296.303,-79.880,178.893,17.205,151.896
C00692=1100.591,296.551,-79.911,178.897,17.207,151.896
C00693=1100.597,296.799,-79.941,178.900,17.209,151.896
C00694=1100.603,297.048,-79.971,178.904,17.211,151.896
C00695=1100.609,297.296,-80.001,178.907,17.212,151.895
C00696=1100.615,297.543,-80.032,178.910,17.214,151.895
C00697=1100.621,297.792,-80.061,178.914,17.216,151.895
C00698=1100.626,298.040,-80.092,178.917,17.218,151.895
C00699=1100.631,298.288,-80.123,178.921,17.220,151.894
C00700=1100.637,298.536,-80.153,178.924,17.221,151.894
C00701=1100.643,298.784,-80.182,178.927,17.223,151.894
C00702=1100.648,299.032,-80.213,178.931,17.225,151.894
C00703=1100.654,299.280,-80.244,178.934,17.227,151.893
C00704=1100.659,299.528,-80.274,178.938,17.228,151.893
C00705=1100.665,299.776,-80.304,178.941,17.230,151.893
C00706=1100.670,300.024,-80.335,178.945,17.233,151.893
C00707=1100.676,300.272,-80.365,178.948,17.235,151.892
C00708=1100.682,300.520,-80.395,178.951,17.236,151.892
C00709=1100.687,300.768,-80.426,178.954,17.238,151.892
C00710=1100.693,301.016,-80.457,178.958,17.240,151.892
C00711=1100.698,301.264,-80.487,178.961,17.242,151.891
C00712=1100.704,301.512,-80.518,178.965,17.244,151.891
C00713=1100.709,301.760,-80.548,178.968,17.246,151.891
C00714=1100.714,302.008,-80.579,178.972,17.247,151.891
C00715=1100.720,302.256,-80.610,178.975,17.249,151.891
C00716=1100.730,302.638,-80.657,178.980,17.253,151.890
C00717=1100.737,303.020,-80.704,178.985,17.255,151.890
C00718=1100.747,303.403,-80.752,178.991,17.258,151.890
C00719=1100.755,303.784,-80.799,178.996,17.261,151.889
C00720=1100.760,304.032,-80.830,178.999,17.263,151.889
C00721=1100.766,304.280,-80.860,179.003,17.265,151.889
C00722=1100.772,304.529,-80.891,179.005,17.267,151.889
C00723=1100.778,304.777,-80.922,179.009,17.269,151.888
C00724=1100.783,305.024,-80.952,179.012,17.271,151.888
C00725=1100.789,305.273,-80.983,179.016,17.273,151.888
C00726=1100.795,305.520,-81.014,179.019,17.274,151.888
C00727=1100.800,305.768,-81.045,179.023,17.276,151.887
C00728=1100.806,306.016,-81.076,179.026,17.278,151.887
C00729=1100.811,306.265,-81.107,179.030,17.280,151.887
C00730=1100.817,306.512,-81.137,179.033,17.282,151.887
C00731=1100.822,306.760,-81.169,179.037,17.284,151.887
C00732=1100.828,307.008,-81.199,179.040,17.286,151.886
C00733=1100.834,307.257,-81.230,179.043,17.288,151.886
C00734=1100.840,307.504,-81.261,179.046,17.290,151.886
C00735=1100.845,307.752,-81.292,179.050,17.292,151.886
C00736=1100.851,308.000,-81.323,179.053,17.294,151.886
C00737=1100.857,308.249,-81.354,179.056,17.296,151.885
C00738=1100.863,308.496,-81.385,179.060,17.298,151.885
C00739=1100.868,308.744,-81.416,179.063,17.300,151.885
C00740=1100.875,308.992,-81.447,179.067,17.302,151.885
C00741=1100.880,309.240,-81.478,179.070,17.304,151.885
C00742=1100.885,309.488,-81.509,179.074,17.306,151.884
C00743=1100.891,309.736,-81.541,179.077,17.308,151.884
C00744=1100.897,309.984,-81.572,179.080,17.310,151.884
C00745=1100.903,310.231,-81.603,179.084,17.312,151.884
C00746=1100.908,310.480,-81.634,179.087,17.314,151.884
C00747=1100.914,310.728,-81.664,179.091,17.316,151.883
C00748=1100.920,310.975,-81.696,179.094,17.318,151.883
C00749=1100.925,311.224,-81.727,179.097,17.320,151.883
C00750=1100.931,311.471,-81.758,179.100,17.322,151.883
C00751=1100.936,311.720,-81.789,179.104,17.324,151.883
C00752=1100.943,311.968,-81.821,179.107,17.326,151.882
C00753=1100.949,312.215,-81.852,179.110,17.328,151.882
C00754=1100.954,312.464,-81.884,179.114,17.330,151.882
C00755=1100.960,312.711,-81.915,179.117,17.332,151.882
C00756=1100.965,312.959,-81.946,179.120,17.334,151.882
C00757=1100.971,313.207,-81.978,179.124,17.336,151.882
C00758=1100.978,313.455,-82.009,179.127,17.338,151.881
C00759=1100.983,313.703,-82.040,179.131,17.340,151.881
C00760=1100.989,313.951,-82.072,179.134,17.342,151.881
C00761=1100.995,314.199,-82.103,179.138,17.345,151.881
C00762=1101.000,314.447,-82.134,179.141,17.347,151.881
C00763=1101.006,314.695,-82.166,179.144,17.349,151.881
C00764=1101.012,314.943,-82.198,179.148,17.351,151.880
C00765=1101.018,315.191,-82.228,179.151,17.353,151.880
C00766=1101.024,315.439,-82.260,179.154,17.355,151.880
C00767=1101.029,315.686,-82.292,179.158,17.357,151.880
C00768=1101.038,316.071,-82.341,179.163,17.361,151.880
C00769=1101.046,316.456,-82.390,179.168,17.364,151.880
C00770=1101.055,316.841,-82.439,179.173,17.367,151.879
C00771=1101.063,317.225,-82.488,179.178,17.371,151.879
C00772=1101.069,317.473,-82.519,179.181,17.374,151.879
C00773=1101.075,317.721,-82.551,179.185,17.376,151.879
C00774=1101.080,317.969,-82.583,179.188,17.378,151.879
C00775=1101.086,318.217,-82.615,179.191,17.380,151.879
C00776=1101.092,318.464,-82.647,179.195,17.383,151.879
C00777=1101.098,318.713,-82.679,179.198,17.385,151.879
C00778=1101.103,318.961,-82.710,179.201,17.387,151.878
C00779=1101.107,319.209,-82.742,179.205,17.389,151.878
C00780=1101.113,319.457,-82.774,179.208,17.392,151.878
C00781=1101.119,319.704,-82.806,179.211,17.394,151.878
C00782=1101.125,319.952,-82.838,179.214,17.396,151.878
C00783=1101.130,320.200,-82.869,179.217,17.399,151.878
C00784=1101.136,320.448,-82.901,179.221,17.401,151.878
C00785=1101.141,320.696,-82.933,179.224,17.403,151.878
C00786=1101.147,320.944,-82.965,179.227,17.405,151.878
C00787=1101.153,321.192,-82.997,179.231,17.408,151.878
C00788=1101.159,321.440,-83.029,179.234,17.410,151.878
C00789=1101.164,321.688,-83.061,179.237,17.412,151.877
C00790=1101.170,321.935,-83.094,179.240,17.415,151.877
C00791=1101.176,322.183,-83.126,179.243,17.417,151.877
C00792=1101.181,322.431,-83.158,179.248,17.420,151.877
C00793=1101.187,322.679,-83.190,179.251,17.422,151.877
C00794=1101.193,322.927,-83.221,179.254,17.425,151.877
C00795=1101.198,323.175,-83.253,179.257,17.427,151.877
C00796=1101.204,323.423,-83.286,179.261,17.429,151.877
C00797=1101.209,323.670,-83.318,179.264,17.432,151.877
C00798=1101.215,323.918,-83.350,179.267,17.434,151.877
C00799=1101.221,324.166,-83.382,179.270,17.436,151.877
C00800=1101.227,324.414,-83.414,179.273,17.439,151.876
C00801=1101.232,324.663,-83.447,179.277,17.441,151.876
C00802=1101.238,324.909,-83.479,179.280,17.443,151.876
C00803=1101.244,325.158,-83.511,179.283,17.445,151.876
C00804=1101.250,325.406,-83.543,179.286,17.448,151.876
C00805=1101.255,325.653,-83.575,179.289,17.450,151.876
C00806=1101.261,325.901,-83.608,179.294,17.453,151.876
C00807=1101.267,326.150,-83.640,179.297,17.455,151.876
C00808=1101.272,326.396,-83.672,179.300,17.458,151.876
C00809=1101.278,326.645,-83.704,179.303,17.460,151.876
C00810=1101.284,326.893,-83.737,179.306,17.463,151.876
C00811=1101.289,327.140,-83.769,179.310,17.465,151.876
C00812=1101.295,327.388,-83.801,179.313,17.467,151.876
C00813=1101.301,327.636,-83.835,179.316,17.470,151.876
C00814=1101.307,327.884,-83.867,179.319,17.472,151.876
C00815=1101.312,328.132,-83.898,179.323,17.475,151.876
C00816=1101.318,328.380,-83.931,179.326,17.478,151.875
C00817=1101.324,328.628,-83.964,179.329,17.480,151.875
C00818=1101.330,328.876,-83.997,179.333,17.482,151.875
C00819=1101.335,329.123,-84.028,179.336,17.485,151.875
C00820=1101.344,329.501,-84.079,179.341,17.488,151.875
C00821=1101.353,329.879,-84.128,179.346,17.493,151.875
C00822=1101.362,330.256,-84.178,179.351,17.496,151.875
C00823=1101.371,330.634,-84.227,179.356,17.500,151.875
C00824=1101.376,330.882,-84.260,179.359,17.503,151.875
C00825=1101.382,331.129,-84.293,179.363,17.506,151.875
C00826=1101.388,331.377,-84.325,179.366,17.508,151.875
C00827=1101.394,331.625,-84.358,179.369,17.511,151.875
C00828=1101.400,331.872,-84.391,179.372,17.513,151.875
C00829=1101.405,332.121,-84.423,179.375,17.516,151.875
C00830=1101.411,332.368,-84.456,179.378,17.518,151.875
C00831=1101.417,332.616,-84.489,179.382,17.521,151.875
C00832=1101.423,332.864,-84.522,179.385,17.524,151.875
C00833=1101.428,333.112,-84.554,179.388,17.526,151.875
C00834=1101.433,333.360,-84.588,179.391,17.529,151.875
C00835=1101.440,333.607,-84.620,179.395,17.531,151.875
C00836=1101.445,333.855,-84.654,179.397,17.534,151.875
C00837=1101.451,334.103,-84.686,179.401,17.537,151.875
C00838=1101.457,334.351,-84.719,179.405,17.540,151.875
C00839=1101.462,334.598,-84.752,179.408,17.542,151.875
C00840=1101.468,334.846,-84.785,179.411,17.545,151.875
C00841=1101.473,335.094,-84.818,179.414,17.547,151.875
C00842=1101.479,335.342,-84.851,179.418,17.551,151.875
C00843=1101.485,335.590,-84.883,179.420,17.553,151.875
C00844=1101.491,335.838,-84.917,179.424,17.556,151.875
C00845=1101.495,336.085,-84.950,179.426,17.559,151.875
C00846=1101.502,336.333,-84.983,179.430,17.562,151.875
C00847=1101.507,336.581,-85.016,179.434,17.564,151.875
C00848=1101.513,336.828,-85.049,179.436,17.567,151.875
C00849=1101.519,337.076,-85.082,179.440,17.570,151.875
C00850=1101.525,337.324,-85.115,179.443,17.573,151.875
C00851=1101.530,337.572,-85.149,179.446,17.576,151.875
C00852=1101.537,337.819,-85.181,179.449,17.578,151.875
C00853=1101.542,338.067,-85.215,179.452,17.581,151.875
C00854=1101.548,338.315,-85.248,179.455,17.584,151.876
C00855=1101.553,338.563,-85.281,179.459,17.587,151.876
C00856=1101.560,338.811,-85.314,179.462,17.590,151.876
C00857=1101.564,339.058,-85.347,179.465,17.592,151.876
C00858=1101.570,339.305,-85.381,179.469,17.596,151.876
C00859=1101.576,339.553,-85.414,179.472,17.598,151.876
C00860=1101.581,339.801,-85.448,179.475,17.601,151.876
C00861=1101.587,340.049,-85.481,179.478,17.604,151.876
C00862=1101.593,340.297,-85.515,179.482,17.607,151.876
C00863=1101.599,340.544,-85.547,179.485,17.610,151.876
C00864=1101.605,340.792,-85.581,179.487,17.613,151.876
C00865=1101.610,341.040,-85.615,179.491,17.616,151.876
C00866=1101.616,341.288,-85.648,179.494,17.619,151.876
C00867=1101.621,341.535,-85.681,179.497,17.622,151.876
C00868=1101.627,341.783,-85.715,179.500,17.624,151.877
C00869=1101.633,342.031,-85.749,179.504,17.628,151.877
C00870=1101.638,342.279,-85.782,179.507,17.630,151.877
C00871=1101.644,342.526,-85.815,179.510,17.633,151.877
C00872=1101.653,342.898,-85.866,179.515,17.638,151.877
C00873=1101.661,343.270,-85.916,179.519,17.643,151.877
C00874=1101.670,343.641,-85.967,179.524,17.647,151.877
C00875=1101.679,344.012,-86.017,179.529,17.651,151.877
C00876=1101.684,344.260,-86.050,179.532,17.655,151.878
C00877=1101.690,344.508,-86.084,179.535,17.658,151.878
C00878=1101.696,344.755,-86.118,179.538,17.661,151.878
C00879=1101.701,345.003,-86.151,179.542,17.664,151.878
C00880=1101.707,345.250,-86.185,179.545,17.667,151.878
C00881=1101.712,345.498,-86.219,179.548,17.670,151.878
C00882=1101.718,345.746,-86.253,179.551,17.673,151.878
C00883=1101.724,345.993,-86.286,179.554,17.676,151.879
C00884=1101.729,346.241,-86.320,179.557,17.679,151.879
C00885=1101.735,346.489,-86.354,179.561,17.683,151.879
C00886=1101.741,346.737,-86.388,179.564,17.685,151.879
C00887=1101.747,346.984,-86.422,179.566,17.688,151.879
C00888=1101.753,347.232,-86.456,179.570,17.692,151.879
C00889=1101.758,347.479,-86.490,179.573,17.695,151.879
C00890=1101.763,347.727,-86.524,179.576,17.699,151.880
C00891=1101.769,347.975,-86.558,179.579,17.701,151.880
C00892=1101.775,348.222,-86.592,179.582,17.704,151.880
C00893=1101.781,348.470,-86.625,179.585,17.708,151.880
C00894=1101.786,348.717,-86.660,179.588,17.711,151.880
C00895=1101.792,348.965,-86.694,179.591,17.714,151.880
C00896=1101.798,349.213,-86.728,179.595,17.717,151.881
C00897=1101.804,349.461,-86.761,179.597,17.721,151.881
C00898=1101.810,349.708,-86.796,179.601,17.724,151.881
C00899=1101.815,349.955,-86.830,179.604,17.727,151.881
C00900=1101.821,350.203,-86.864,179.607,17.731,151.881
C00901=1101.826,350.451,-86.898,179.610,17.734,151.882
C00902=1101.831,350.698,-86.932,179.613,17.737,151.882
C00903=1101.838,350.946,-86.967,179.617,17.741,151.882
C00904=1101.844,351.193,-87.001,179.619,17.743,151.882
C00905=1101.849,351.441,-87.035,179.623,17.747,151.882
C00906=1101.855,351.688,-87.069,179.626,17.750,151.883
C00907=1101.860,351.936,-87.103,179.629,17.754,151.883
C00908=1101.867,352.184,-87.137,179.632,17.757,151.883
C00909=1101.872,352.432,-87.172,179.635,17.760,151.883
C00910=1101.878,352.679,-87.206,179.638,17.764,151.883
C00911=1101.883,352.926,-87.240,179.641,17.767,151.884
C00912=1101.889,353.174,-87.275,179.644,17.771,151.884
C00913=1101.895,353.422,-87.309,179.647,17.774,151.884
C00914=1101.901,353.669,-87.343,179.650,17.778,151.884
C00915=1101.906,353.917,-87.378,179.653,17.781,151.884
C00916=1101.912,354.164,-87.412,179.657,17.784,151.885
C00917=1101.917,354.412,-87.446,179.659,17.788,151.885
C00918=1101.923,354.660,-87.481,179.663,17.791,151.885
C00919=1101.929,354.907,-87.515,179.666,17.795,151.885
C00920=1101.934,355.155,-87.549,179.669,17.798,151.886
C00921=1101.940,355.402,-87.585,179.672,17.802,151.886
C00922=1101.946,355.650,-87.619,179.675,17.805,151.886
C00923=1101.951,355.897,-87.654,179.678,17.808,151.886
C00924=1101.960,356.271,-87.705,179.683,17.814,151.887
C00925=1101.969,356.644,-87.758,179.687,17.820,151.887
C00926=1101.977,357.019,-87.810,179.691,17.824,151.888
C00927=1101.986,357.392,-87.863,179.696,17.830,151.888
C00928=1101.991,357.639,-87.897,179.699,17.834,151.889
C00929=1101.997,357.888,-87.932,179.702,17.837,151.889
C00930=1102.003,358.134,-87.967,179.705,17.841,151.889
C00931=1102.008,358.382,-88.001,179.708,17.844,151.889
C00932=1102.015,358.630,-88.036,179.711,17.848,151.890
C00933=1102.020,358.877,-88.071,179.714,17.852,151.890
C00934=1102.025,359.124,-88.106,179.717,17.855,151.890
C00935=1102.032,359.372,-88.140,179.720,17.859,151.891
C00936=1102.037,359.619,-88.176,179.723,17.863,151.891
C00937=1102.043,359.867,-88.210,179.726,17.866,151.891
C00938=1102.049,360.115,-88.245,179.729,17.870,151.891
C00939=1102.054,360.362,-88.280,179.733,17.874,151.892
C00940=1102.061,360.610,-88.314,179.735,17.877,151.892
C00941=1102.066,360.857,-88.350,179.738,17.881,151.892
C00942=1102.071,361.104,-88.384,179.741,17.885,151.893
C00943=1102.077,361.352,-88.420,179.744,17.888,151.893
C00944=1102.083,361.599,-88.454,179.747,17.892,151.893
C00945=1102.089,361.846,-88.490,179.750,17.896,151.894
C00946=1102.094,362.095,-88.525,179.754,17.900,151.894
C00947=1102.100,362.342,-88.560,179.756,17.904,151.895
C00948=1102.106,362.589,-88.594,179.759,17.907,151.895
C00949=1102.112,362.837,-88.630,179.762,17.911,151.895
C00950=1102.117,363.084,-88.665,179.765,17.915,151.896
C00951=1102.123,363.332,-88.700,179.768,17.919,151.896
C00952=1102.129,363.578,-88.735,179.771,17.923,151.896
C00953=1102.135,363.826,-88.771,179.774,17.927,151.897
C00954=1102.140,364.074,-88.805,179.777,17.930,151.897
C00955=1102.146,364.321,-88.841,179.780,17.934,151.897
C00956=1102.152,364.568,-88.876,179.783,17.938,151.898
C00957=1102.158,364.816,-88.910,179.785,17.942,151.898
C00958=1102.164,365.063,-88.946,179.789,17.946,151.898
C00959=1102.169,365.310,-88.981,179.791,17.950,151.899
C00960=1102.175,365.559,-89.016,179.794,17.954,151.899
C00961=1102.180,365.806,-89.052,179.798,17.958,151.900
C00962=1102.186,366.053,-89.088,179.800,17.962,151.900
C00963=1102.192,366.300,-89.123,179.803,17.966,151.901
C00964=1102.197,366.547,-89.158,179.806,17.970,151.901
C00965=1102.203,366.795,-89.194,179.809,17.974,151.901
C00966=1102.208,367.042,-89.229,179.812,17.978,151.902
C00967=1102.214,367.290,-89.264,179.815,17.982,151.902
C00968=1102.220,367.537,-89.300,179.818,17.986,151.903
C00969=1102.226,367.785,-89.336,179.821,17.990,151.903
C00970=1102.231,368.032,-89.371,179.824,17.994,151.904
C00971=1102.237,368.279,-89.407,179.826,17.998,151.904
C00972=1102.243,368.526,-89.442,179.829,18.002,151.904
C00973=1102.249,368.774,-89.478,179.833,18.007,151.905
C00974=1102.254,369.021,-89.513,179.835,18.010,151.905
C00975=1102.260,369.269,-89.549,179.838,18.014,151.906
C00976=1102.269,369.657,-89.604,179.842,18.021,151.907
C00977=1102.278,370.046,-89.661,179.847,18.028,151.907
C00978=1102.287,370.434,-89.717,179.851,18.034,151.908
C00979=1102.296,370.823,-89.773,179.856,18.041,151.909
C00980=1102.301,371.070,-89.808,179.859,18.045,151.909
C00981=1102.307,371.318,-89.844,179.862,18.049,151.910
C00982=1102.313,371.565,-89.880,179.865,18.054,151.910
C00983=1102.319,371.813,-89.915,179.868,18.058,151.911
C00984=1102.325,372.060,-89.951,179.870,18.062,151.911
C00985=1102.330,372.307,-89.987,179.873,18.066,151.912
C00986=1102.336,372.554,-90.023,179.876,18.071,151.912
C00987=1102.341,372.802,-90.059,179.879,18.075,151.913
C00988=1102.347,373.049,-90.095,179.881,18.079,151.913
C00989=1102.353,373.297,-90.130,179.884,18.084,151.914
C00990=1102.359,373.543,-90.166,179.887,18.088,151.914
C00991=1102.365,373.791,-90.202,179.891,18.092,151.915
C00992=1102.371,374.039,-90.238,179.893,18.096,151.915
C00993=1102.376,374.285,-90.274,179.896,18.101,151.916
C00994=1102.382,374.533,-90.310,179.899,18.105,151.916
C00995=1102.387,374.780,-90.346,179.902,18.110,151.917
C00996=1102.393,375.027,-90.383,179.904,18.114,151.918
C00997=1102.399,375.275,-90.418,179.907,18.118,151.918
C00998=1102.405,375.521,-90.454,179.910,18.123,151.919
C00999=1102.410,375.769,-90.491,179.913,18.128,151.919
C01000=1102.416,376.017,-90.526,179.915,18.133,151.920
C01001=1102.422,376.263,-90.563,179.918,18.137,151.920
C01002=1102.427,376.511,-90.599,179.920,18.141,151.921
C01003=1102.433,376.758,-90.635,179.924,18.146,151.922
C01004=1102.438,377.006,-90.671,179.926,18.150,151.922
C01005=1102.444,377.253,-90.708,179.929,18.155,151.923
C01006=1102.450,377.500,-90.743,179.932,18.160,151.923
C01007=1102.455,377.747,-90.780,179.934,18.164,151.924
C01008=1102.462,377.994,-90.817,179.937,18.168,151.925
C01009=1102.467,378.241,-90.853,179.940,18.173,151.925
C01010=1102.473,378.488,-90.889,179.943,18.178,151.926
C01011=1102.479,378.736,-90.925,179.946,18.183,151.926
C01012=1102.484,378.983,-90.961,179.949,18.188,151.927
C01013=1102.490,379.230,-90.998,179.951,18.192,151.928
C01014=1102.495,379.478,-91.034,179.954,18.196,151.928
C01015=1102.502,379.725,-91.071,179.956,18.201,151.929
C01016=1102.507,379.971,-91.107,179.959,18.206,151.930
C01017=1102.513,380.219,-91.143,179.962,18.211,151.930
C01018=1102.518,380.467,-91.180,179.965,18.216,151.931
C01019=1102.525,380.714,-91.216,179.967,18.221,151.932
C01020=1102.530,380.960,-91.253,179.970,18.225,151.932
C01021=1102.536,381.208,-91.289,179.973,18.230,151.933
C01022=1102.541,381.455,-91.326,179.975,18.234,151.934
C01023=1102.548,381.702,-91.362,179.978,18.239,151.934
C01024=1102.553,381.950,-91.399,179.981,18.244,151.935
C01025=1102.559,382.196,-91.435,179.983,18.249,151.935
C01026=1102.565,382.443,-91.473,179.986,18.254,151.936
C01027=1102.571,382.690,-91.509,179.989,18.259,151.937
C01028=1102.580,383.106,-91.570,179.993,18.267,151.938
C01029=1102.590,383.522,-91.632,179.998,18.276,151.939
C01030=1102.599,383.937,-91.694,-179.998,18.284,151.940
C01031=1102.608,384.353,-91.756,-179.993,18.292,151.942
C01032=1102.614,384.600,-91.793,-179.991,18.297,151.942
C01033=1102.620,384.847,-91.829,-179.988,18.302,151.943
C01034=1102.626,385.095,-91.866,-179.985,18.307,151.944
C01035=1102.632,385.342,-91.903,-179.983,18.312,151.945
C01036=1102.637,385.589,-91.940,-179.980,18.317,151.945
C01037=1102.643,385.836,-91.976,-179.977,18.322,151.946
C01038=1102.648,386.083,-92.013,-179.975,18.327,151.947
C01039=1102.654,386.330,-92.051,-179.972,18.333,151.948
C01040=1102.660,386.577,-92.088,-179.970,18.338,151.948
C01041=1102.666,386.824,-92.125,-179.967,18.343,151.949
C01042=1102.671,387.071,-92.161,-179.965,18.348,151.950
C01043=1102.677,387.318,-92.198,-179.962,18.353,151.951
C01044=1102.683,387.565,-92.235,-179.959,18.358,151.952
C01045=1102.688,387.812,-92.273,-179.957,18.363,151.952
C01046=1102.694,388.060,-92.310,-179.953,18.370,151.953
C01047=1102.700,388.307,-92.347,-179.951,18.375,151.954
C01048=1102.706,388.553,-92.384,-179.948,18.380,151.955
C01049=1102.712,388.801,-92.422,-179.946,18.385,151.956
C01050=1102.717,389.048,-92.459,-179.943,18.390,151.956
C01051=1102.723,389.295,-92.496,-179.941,18.396,151.957
C01052=1102.728,389.542,-92.533,-179.938,18.401,151.958
C01053=1102.734,389.789,-92.570,-179.936,18.406,151.959
C01054=1102.741,390.035,-92.607,-179.933,18.411,151.960
C01055=1102.746,390.283,-92.644,-179.931,18.417,151.961
C01056=1102.752,390.530,-92.681,-179.928,18.422,151.961
C01057=1102.758,390.777,-92.719,-179.926,18.427,151.962
C01058=1102.763,391.024,-92.756,-179.923,18.433,151.963
C01059=1102.769,391.271,-92.794,-179.921,18.438,151.964
C01060=1102.775,391.518,-92.831,-179.917,18.444,151.965
C01061=1102.781,391.765,-92.869,-179.915,18.450,151.966
C01062=1102.786,392.012,-92.906,-179.913,18.455,151.967
C01063=1102.792,392.259,-92.943,-179.910,18.460,151.968
C01064=1102.798,392.507,-92.981,-179.908,18.466,151.969
C01065=1102.804,392.753,-93.018,-179.905,18.471,151.969
C01066=1102.810,393.001,-93.056,-179.903,18.477,151.970
C01067=1102.816,393.248,-93.093,-179.901,18.482,151.971
C01068=1102.821,393.495,-93.130,-179.897,18.488,151.972
C01069=1102.827,393.742,-93.168,-179.895,18.494,151.973
C01070=1102.833,393.989,-93.206,-179.893,18.499,151.974
C01071=1102.839,394.236,-93.243,-179.890,18.505,151.975
C01072=1102.844,394.483,-93.281,-179.888,18.511,151.976
C01073=1102.850,394.730,-93.319,-179.886,18.516,151.977
C01074=1102.855,394.977,-93.356,-179.883,18.522,151.978
C01075=1102.861,395.224,-93.394,-179.880,18.528,151.979
C01076=1102.867,395.471,-93.432,-179.878,18.534,151.980
C01077=1102.873,395.718,-93.469,-179.876,18.540,151.981
C01078=1102.878,395.965,-93.507,-179.873,18.545,151.982
C01079=1102.884,396.212,-93.545,-179.871,18.551,151.983
C01080=1102.890,396.426,-93.578,-179.869,18.556,151.984
C01081=1102.894,396.641,-93.610,-179.867,18.561,151.984
C01082=1102.899,396.854,-93.643,-179.864,18.566,151.985
C01083=1102.904,397.068,-93.676,-179.862,18.572,151.986
C01084=1102.909,397.282,-93.709,-179.860,18.577,151.987
C01085=1102.914,397.496,-93.741,-179.858,18.582,151.988
C01086=1102.919,397.710,-93.774,-179.856,18.587,151.989
C01087=1102.924,397.923,-93.807,-179.854,18.592,151.990
C01088=1102.930,398.171,-93.845,-179.851,18.598,151.991
C01089=1102.935,398.418,-93.883,-179.849,18.604,151.992
C01090=1102.941,398.665,-93.921,-179.847,18.610,151.993
C01091=1102.947,398.911,-93.959,-179.844,18.616,151.994
C01092=1102.952,399.159,-93.997,-179.842,18.622,151.995
C01093=1102.959,399.407,-94.035,-179.840,18.628,151.996
C01094=1102.964,399.653,-94.073,-179.837,18.634,151.997
C01095=1102.970,399.900,-94.111,-179.835,18.640,151.998
C01096=1102.975,400.147,-94.149,-179.833,18.646,151.999
C01097=1102.981,400.394,-94.187,-179.831,18.652,152.000
C01098=1102.987,400.641,-94.226,-179.828,18.659,152.001
C01099=1102.993,400.888,-94.264,-179.826,18.665,152.003
C01100=1102.999,401.135,-94.302,-179.824,18.671,152.004
C01101=1103.004,401.381,-94.340,-179.821,18.678,152.005
C01102=1103.010,401.629,-94.378,-179.819,18.684,152.006
C01103=1103.016,401.876,-94.416,-179.817,18.690,152.007
C01104=1103.021,402.123,-94.454,-179.814,18.696,152.008
C01105=1103.027,402.370,-94.492,-179.812,18.703,152.009
C01106=1103.033,402.617,-94.532,-179.809,18.709,152.010
C01107=1103.039,402.864,-94.569,-179.807,18.715,152.012
C01108=1103.044,403.111,-94.608,-179.805,18.721,152.013
C01109=1103.050,403.358,-94.646,-179.802,18.728,152.014
C01110=1103.056,403.605,-94.684,-179.800,18.734,152.015
C01111=1103.061,403.852,-94.723,-179.797,18.741,152.016
C01112=1103.067,404.098,-94.761,-179.795,18.747,152.017
C01113=1103.073,404.346,-94.800,-179.794,18.754,152.019
C01114=1103.079,404.592,-94.838,-179.791,18.760,152.020
C01115=1103.085,404.839,-94.877,-179.789,18.767,152.021
C01116=1103.090,405.087,-94.915,-179.786,18.774,152.022
C01117=1103.097,405.333,-94.954,-179.784,18.780,152.023
C01118=1103.102,405.580,-94.992,-179.781,18.787,152.025
C01119=1103.108,405.827,-95.032,-179.780,18.793,152.026
C01120=1103.114,406.074,-95.069,-179.777,18.800,152.027
C01121=1103.119,406.322,-95.108,-179.775,18.806,152.028
C01122=1103.125,406.568,-95.147,-179.773,18.814,152.030
C01123=1103.131,406.815,-95.185,-179.771,18.820,152.031
C01124=1103.137,407.062,-95.224,-179.768,18.827,152.032
C01125=1103.142,407.309,-95.263,-179.766,18.833,152.033
C01126=1103.148,407.556,-95.302,-179.764,18.841,152.035
C01127=1103.153,407.803,-95.340,-179.762,18.847,152.036
C01128=1103.159,408.050,-95.379,-179.759,18.854,152.037
C01129=1103.166,408.297,-95.418,-179.758,18.861,152.039
C01130=1103.171,408.544,-95.457,-179.755,18.868,152.040
C01131=1103.176,408.790,-95.496,-179.752,18.875,152.041
C01132=1103.182,409.038,-95.534,-179.751,18.882,152.043
C01133=1103.187,409.284,-95.574,-179.748,18.889,152.044
C01134=1103.194,409.532,-95.613,-179.746,18.895,152.045
C01135=1103.199,409.778,-95.651,-179.744,18.903,152.047
C01136=1103.205,409.992,-95.685,-179.742,18.909,152.048
C01137=1103.209,410.206,-95.718,-179.740,18.915,152.049
C01138=1103.215,410.420,-95.753,-179.738,18.921,152.050
C01139=1103.219,410.634,-95.786,-179.737,18.927,152.051
C01140=1103.224,410.847,-95.820,-179.735,18.933,152.053
C01141=1103.229,411.062,-95.854,-179.733,18.939,152.054
C01142=1103.234,411.275,-95.888,-179.731,18.946,152.055
C01143=1103.239,411.490,-95.921,-179.729,18.952,152.056
C01144=1103.245,411.736,-95.960,-179.727,18.960,152.058
C01145=1103.251,411.983,-96.000,-179.725,18.966,152.059
C01146=1103.256,412.230,-96.039,-179.723,18.974,152.061
C01147=1103.262,412.477,-96.078,-179.720,18.981,152.062
C01148=1103.268,412.723,-96.117,-179.718,18.989,152.063
C01149=1103.274,412.970,-96.157,-179.716,18.996,152.065
C01150=1103.279,413.217,-96.196,-179.714,19.003,152.066
C01151=1103.285,413.464,-96.235,-179.712,19.011,152.068
C01152=1103.291,413.710,-96.274,-179.710,19.018,152.069
C01153=1103.297,413.957,-96.314,-179.708,19.025,152.071
C01154=1103.302,414.204,-96.353,-179.706,19.033,152.072
C01155=1103.308,414.451,-96.392,-179.703,19.041,152.074
C01156=1103.314,414.698,-96.432,-179.701,19.048,152.075
C01157=1103.320,414.945,-96.471,-179.699,19.055,152.077
C01158=1103.326,415.192,-96.510,-179.697,19.063,152.078
C01159=1103.331,415.438,-96.549,-179.695,19.070,152.080
C01160=1103.338,415.685,-96.589,-179.693,19.078,152.081
C01161=1103.343,415.933,-96.629,-179.690,19.086,152.083
C01162=1103.348,416.179,-96.668,-179.689,19.093,152.084
C01163=1103.355,416.426,-96.708,-179.687,19.101,152.086
C01164=1103.361,416.673,-96.747,-179.684,19.108,152.087
C01165=1103.366,416.919,-96.786,-179.682,19.116,152.089
C01166=1103.372,417.166,-96.826,-179.680,19.124,152.090
C01167=1103.377,417.412,-96.866,-179.678,19.132,152.092
C01168=1103.383,417.660,-96.906,-179.676,19.140,152.094
C01169=1103.389,417.906,-96.945,-179.675,19.148,152.095
C01170=1103.395,418.153,-96.984,-179.673,19.156,152.097
C01171=1103.401,418.400,-97.025,-179.670,19.164,152.099
C01172=1103.406,418.646,-97.064,-179.668,19.172,152.100
C01173=1103.412,418.893,-97.104,-179.666,19.180,152.102
C01174=1103.418,419.140,-97.144,-179.664,19.188,152.103
C01175=1103.423,419.387,-97.183,-179.662,19.196,152.105
C01176=1103.430,419.633,-97.223,-179.660,19.204,152.107
C01177=1103.434,419.880,-97.263,-179.658,19.212,152.108
C01178=1103.441,420.127,-97.303,-179.656,19.220,152.110
C01179=1103.447,420.374,-97.343,-179.654,19.228,152.112
C01180=1103.453,420.621,-97.383,-179.652,19.236,152.113
C01181=1103.458,420.867,-97.422,-179.650,19.244,152.115
C01182=1103.464,421.114,-97.463,-179.648,19.252,152.117
C01183=1103.470,421.361,-97.503,-179.646,19.261,152.119
C01184=1103.475,421.607,-97.542,-179.644,19.269,152.120
C01185=1103.482,421.853,-97.583,-179.642,19.277,152.122
C01186=1103.487,422.101,-97.623,-179.640,19.286,152.124
C01187=1103.494,422.347,-97.663,-179.639,19.294,152.126
C01188=1103.498,422.594,-97.702,-179.637,19.302,152.127
C01189=1103.505,422.841,-97.743,-179.635,19.311,152.129
C01190=1103.510,423.087,-97.783,-179.633,19.319,152.131
C01191=1103.517,423.334,-97.823,-179.631,19.328,152.133
C01192=1103.522,423.555,-97.859,-179.629,19.336,152.134
C01193=1103.526,423.775,-97.895,-179.628,19.343,152.136
C01194=1103.531,423.996,-97.931,-179.626,19.351,152.138
C01195=1103.536,424.216,-97.967,-179.624,19.358,152.139
C01196=1103.542,424.437,-98.003,-179.622,19.366,152.141
C01197=1103.547,424.657,-98.039,-179.621,19.374,152.143
C01198=1103.552,424.878,-98.075,-179.619,19.382,152.144
C01199=1103.558,425.099,-98.111,-179.618,19.390,152.146
C01200=1103.563,425.345,-98.151,-179.616,19.398,152.148
C01201=1103.569,425.591,-98.192,-179.614,19.407,152.150
C01202=1103.575,425.838,-98.232,-179.612,19.416,152.152
C01203=1103.580,426.085,-98.273,-179.610,19.425,152.153
C01204=1103.587,426.331,-98.313,-179.608,19.434,152.155
C01205=1103.592,426.577,-98.354,-179.607,19.443,152.157
C01206=1103.597,426.824,-98.394,-179.605,19.451,152.159
C01207=1103.604,427.071,-98.434,-179.602,19.461,152.161
C01208=1103.609,427.318,-98.475,-179.601,19.469,152.163
C01209=1103.615,427.564,-98.516,-179.599,19.479,152.165
C01210=1103.621,427.810,-98.556,-179.598,19.487,152.167
C01211=1103.626,428.057,-98.596,-179.595,19.497,152.169
C01212=1103.632,428.304,-98.637,-179.594,19.506,152.171
C01213=1103.639,428.550,-98.677,-179.592,19.515,152.173
C01214=1103.644,428.797,-98.718,-179.591,19.524,152.175
C01215=1103.650,429.044,-98.759,-179.588,19.534,152.177
C01216=1103.656,429.290,-98.800,-179.587,19.542,152.179
C01217=1103.662,429.537,-98.840,-179.585,19.552,152.181
C01218=1103.667,429.783,-98.881,-179.583,19.561,152.183
C01219=1103.673,430.030,-98.922,-179.582,19.571,152.185
C01220=1103.679,430.276,-98.963,-179.580,19.580,152.187
C01221=1103.684,430.523,-99.004,-179.578,19.590,152.189
C01222=1103.690,430.770,-99.044,-179.577,19.599,152.191
C01223=1103.696,431.016,-99.086,-179.575,19.608,152.194
C01224=1103.702,431.262,-99.126,-179.573,19.618,152.196
C01225=1103.708,431.509,-99.167,-179.572,19.628,152.198
C01226=1103.714,431.755,-99.208,-179.570,19.637,152.200
C01227=1103.720,432.002,-99.249,-179.568,19.647,152.202
C01228=1103.725,432.248,-99.290,-179.567,19.656,152.204
C01229=1103.731,432.494,-99.331,-179.566,19.666,152.206
C01230=1103.737,432.741,-99.372,-179.564,19.676,152.209
C01231=1103.742,432.988,-99.413,-179.562,19.686,152.211
C01232=1103.748,433.234,-99.455,-179.560,19.696,152.213
C01233=1103.754,433.481,-99.495,-179.559,19.705,152.215
C01234=1103.760,433.727,-99.537,-179.557,19.716,152.217
C01235=1103.765,433.974,-99.577,-179.556,19.725,152.220
C01236=1103.771,434.220,-99.619,-179.554,19.736,152.222
C01237=1103.777,434.467,-99.660,-179.552,19.745,152.224
C01238=1103.783,434.713,-99.701,-179.551,19.756,152.227
C01239=1103.789,434.959,-99.743,-179.550,19.766,152.229
C01240=1103.794,435.206,-99.783,-179.547,19.776,152.231
C01241=1103.800,435.452,-99.825,-179.546,19.786,152.233
C01242=1103.806,435.699,-99.867,-179.545,19.796,152.236
C01243=1103.812,435.945,-99.908,-179.544,19.806,152.238
C01244=1103.817,436.192,-99.949,-179.542,19.817,152.240
C01245=1103.823,436.438,-99.991,-179.541,19.827,152.243
C01246=1103.829,436.684,-100.032,-179.539,19.837,152.245
C01247=1103.835,436.930,-100.073,-179.538,19.848,152.248
C01248=1103.844,437.337,-100.142,-179.535,19.865,152.252
C01249=1103.854,437.744,-100.211,-179.533,19.882,152.256
C01250=1103.864,438.151,-100.280,-179.530,19.900,152.260
C01251=1103.873,438.558,-100.347,-179.528,19.917,152.264
C01252=1103.878,438.805,-100.389,-179.527,19.928,152.266
C01253=1103.885,439.052,-100.431,-179.526,19.939,152.269
C01254=1103.891,439.298,-100.473,-179.524,19.950,152.271
C01255=1103.897,439.544,-100.514,-179.523,19.960,152.274
C01256=1103.902,439.791,-100.556,-179.521,19.971,152.276
C01257=1103.908,440.036,-100.598,-179.520,19.982,152.279
C01258=1103.914,440.282,-100.640,-179.519,19.992,152.281
C01259=1103.920,440.529,-100.681,-179.517,20.004,152.284
C01260=1103.925,440.775,-100.723,-179.516,20.015,152.286
C01261=1103.932,441.022,-100.765,-179.515,20.025,152.289
C01262=1103.938,441.268,-100.807,-179.514,20.037,152.291
C01263=1103.943,441.515,-100.849,-179.512,20.048,152.294
C01264=1103.949,441.760,-100.891,-179.511,20.059,152.297
C01265=1103.954,442.007,-100.933,-179.510,20.070,152.299
C01266=1103.960,442.253,-100.974,-179.509,20.082,152.302
C01267=1103.966,442.499,-101.017,-179.507,20.093,152.305
C01268=1103.972,442.746,-101.059,-179.506,20.105,152.307
C01269=1103.978,442.992,-101.101,-179.505,20.115,152.310
C01270=1103.984,443.238,-101.143,-179.504,20.127,152.313
C01271=1103.989,443.484,-101.185,-179.503,20.139,152.316
C01272=1103.995,443.731,-101.227,-179.501,20.150,152.318
C01273=1104.001,443.977,-101.269,-179.501,20.162,152.321
C01274=1104.007,444.223,-101.311,-179.499,20.173,152.324
C01275=1104.013,444.469,-101.354,-179.499,20.185,152.327
C01276=1104.019,444.716,-101.396,-179.499,20.196,152.330
C01277=1104.024,444.961,-101.438,-179.498,20.207,152.332
C01278=1104.030,445.209,-101.481,-179.498,20.219,152.335
C01279=1104.036,445.454,-101.523,-179.499,20.230,152.338
C01280=1104.041,445.701,-101.565,-179.498,20.241,152.341
C01281=1104.048,445.946,-101.607,-179.499,20.252,152.344
C01282=1104.053,446.194,-101.650,-179.499,20.264,152.347
C01283=1104.059,446.439,-101.692,-179.499,20.275,152.350
C01284=1104.065,446.686,-101.734,-179.500,20.286,152.353
C01285=1104.071,446.932,-101.777,-179.501,20.298,152.356
C01286=1104.077,447.178,-101.820,-179.501,20.309,152.359
C01287=1104.082,447.425,-101.862,-179.502,20.320,152.362
C01288=1104.088,447.670,-101.904,-179.503,20.332,152.365
C01289=1104.094,447.917,-101.947,-179.504,20.343,152.368
C01290=1104.099,448.163,-101.989,-179.505,20.354,152.371
C01291=1104.105,448.409,-102.032,-179.507,20.365,152.374
C01292=1104.112,448.656,-102.074,-179.508,20.377,152.377
C01293=1104.117,448.902,-102.116,-179.509,20.388,152.380
C01294=1104.122,449.148,-102.159,-179.511,20.399,152.383
C01295=1104.129,449.395,-102.202,-179.513,20.410,152.386
C01296=1104.135,449.641,-102.244,-179.515,20.421,152.390
C01297=1104.140,449.887,-102.287,-179.516,20.432,152.393
C01298=1104.146,450.133,-102.330,-179.518,20.443,152.396
C01299=1104.152,450.379,-102.372,-179.520,20.455,152.399
C01300=1103.749,450.372,-102.503,-179.594,20.682,152.469
C01301=1103.743,450.126,-102.460,-179.592,20.671,152.466
C01302=1103.737,449.879,-102.419,-179.591,20.660,152.463
C01303=1103.731,449.633,-102.375,-179.588,20.648,152.460
C01304=1103.726,449.387,-102.333,-179.586,20.637,152.457
C01305=1103.720,449.141,-102.290,-179.585,20.626,152.454
C01306=1103.714,448.895,-102.247,-179.584,20.614,152.451
C01307=1103.708,448.648,-102.205,-179.582,20.603,152.447
C01308=1103.702,448.402,-102.162,-179.581,20.592,152.444
C01309=1103.696,448.156,-102.119,-179.580,20.581,152.441
C01310=1103.691,447.910,-102.077,-179.578,20.569,152.438
C01311=1103.685,447.663,-102.034,-179.578,20.558,152.435
C01312=1103.679,447.417,-101.992,-179.577,20.546,152.432
C01313=1103.673,447.171,-101.949,-179.575,20.536,152.429
C01314=1103.667,446.924,-101.907,-179.575,20.524,152.426
C01315=1103.662,446.678,-101.864,-179.574,20.513,152.423
C01316=1103.656,446.433,-101.822,-179.574,20.502,152.420
C01317=1103.650,446.185,-101.779,-179.574,20.490,152.417
C01318=1103.644,445.939,-101.737,-179.573,20.479,152.414
C01319=1103.638,445.694,-101.695,-179.574,20.467,152.411
C01320=1103.633,445.447,-101.652,-179.573,20.456,152.408
C01321=1103.627,445.201,-101.609,-179.573,20.444,152.405
C01322=1103.621,444.955,-101.568,-179.574,20.432,152.402
C01323=1103.615,444.709,-101.525,-179.574,20.421,152.400
C01324=1103.609,444.462,-101.483,-179.575,20.410,152.397
C01325=1103.603,444.216,-101.441,-179.575,20.398,152.394
C01326=1103.598,443.969,-101.398,-179.576,20.386,152.391
C01327=1103.592,443.724,-101.356,-179.577,20.375,152.388
C01328=1103.587,443.477,-101.314,-179.578,20.363,152.386
C01329=1103.580,443.231,-101.272,-179.580,20.352,152.383
C01330=1103.575,442.984,-101.230,-179.580,20.341,152.380
C01331=1103.568,442.739,-101.187,-179.582,20.329,152.377
C01332=1103.563,442.492,-101.145,-179.583,20.317,152.375
C01333=1103.557,442.246,-101.104,-179.584,20.306,152.372
C01334=1103.551,442.000,-101.061,-179.585,20.295,152.369
C01335=1103.545,441.753,-101.019,-179.587,20.283,152.367
C01336=1103.540,441.507,-100.977,-179.588,20.272,152.364
C01337=1103.534,441.261,-100.935,-179.590,20.261,152.361
C01338=1103.528,441.015,-100.894,-179.591,20.250,152.359
C01339=1103.522,440.769,-100.852,-179.592,20.239,152.356
C01340=1103.516,440.522,-100.810,-179.594,20.227,152.354
C01341=1103.510,440.276,-100.767,-179.595,20.216,152.351
C01342=1103.504,440.030,-100.726,-179.596,20.205,152.349
C01343=1103.498,439.783,-100.684,-179.598,20.194,152.346
C01344=1103.493,439.537,-100.643,-179.600,20.183,152.343
C01345=1103.487,439.291,-100.601,-179.600,20.173,152.341
C01346=1103.481,439.044,-100.559,-179.602,20.162,152.338
C01347=1103.475,438.798,-100.517,-179.603,20.151,152.336
C01348=1103.469,438.551,-100.476,-179.605,20.140,152.333
C01349=1103.459,438.150,-100.408,-179.607,20.123,152.329
C01350=1103.450,437.748,-100.340,-179.610,20.105,152.325
C01351=1103.441,437.347,-100.272,-179.612,20.088,152.321
C01352=1103.432,436.945,-100.204,-179.614,20.071,152.318
C01353=1103.426,436.699,-100.163,-179.616,20.060,152.315
C01354=1103.420,436.453,-100.121,-179.617,20.050,152.313
C01355=1103.414,436.207,-100.080,-179.619,20.040,152.310
C01356=1103.408,435.961,-100.039,-179.620,20.029,152.308
C01357=1103.402,435.714,-99.997,-179.622,20.019,152.306
C01358=1103.397,435.467,-99.956,-179.623,20.009,152.303
C01359=1103.391,435.221,-99.914,-179.625,19.998,152.301
C01360=1103.385,434.975,-99.873,-179.627,19.988,152.299
C01361=1103.379,434.729,-99.831,-179.628,19.978,152.296
C01362=1103.373,434.482,-99.791,-179.630,19.967,152.294
C01363=1103.367,434.236,-99.749,-179.631,19.957,152.292
C01364=1103.361,433.989,-99.708,-179.633,19.948,152.290
C01365=1103.356,433.743,-99.667,-179.635,19.937,152.287
C01366=1103.351,433.496,-99.625,-179.636,19.928,152.285
C01367=1103.344,433.250,-99.584,-179.638,19.917,152.283
C01368=1103.338,433.003,-99.543,-179.639,19.908,152.281
C01369=1103.332,432.757,-99.502,-179.641,19.898,152.278
C01370=1103.327,432.510,-99.461,-179.643,19.888,152.276
C01371=1103.321,432.264,-99.420,-179.645,19.878,152.274
C01372=1103.315,432.017,-99.379,-179.646,19.868,152.272
C01373=1103.309,431.771,-99.337,-179.648,19.859,152.270
C01374=1103.304,431.524,-99.297,-179.650,19.849,152.267
C01375=1103.298,431.278,-99.255,-179.651,19.840,152.265
C01376=1103.293,431.032,-99.215,-179.653,19.829,152.263
C01377=1103.287,430.785,-99.174,-179.655,19.820,152.261
C01378=1103.281,430.539,-99.133,-179.656,19.811,152.259
C01379=1103.275,430.292,-99.092,-179.659,19.801,152.257
C01380=1103.269,430.046,-99.052,-179.660,19.791,152.255
C01381=1103.263,429.799,-99.010,-179.662,19.782,152.253
C01382=1103.257,429.552,-98.970,-179.664,19.773,152.251
C01383=1103.252,429.306,-98.929,-179.665,19.763,152.248
C01384=1103.246,429.059,-98.887,-179.667,19.754,152.247
C01385=1103.239,428.813,-98.847,-179.669,19.744,152.244
C01386=1103.234,428.567,-98.807,-179.671,19.735,152.242
C01387=1103.229,428.320,-98.766,-179.672,19.726,152.240
C01388=1103.223,428.073,-98.725,-179.674,19.717,152.238
C01389=1103.216,427.827,-98.685,-179.676,19.708,152.236
C01390=1103.211,427.580,-98.644,-179.678,19.698,152.234
C01391=1103.205,427.334,-98.603,-179.680,19.690,152.232
C01392=1103.199,427.087,-98.563,-179.681,19.681,152.230
C01393=1103.193,426.840,-98.522,-179.684,19.671,152.229
C01394=1103.188,426.594,-98.482,-179.685,19.662,152.227
C01395=1103.182,426.348,-98.442,-179.687,19.654,152.225
C01396=1103.176,426.101,-98.401,-179.689,19.644,152.223
C01397=1103.170,425.854,-98.360,-179.690,19.636,152.221
C01398=1103.164,425.607,-98.320,-179.693,19.626,152.219
C01399=1103.159,425.361,-98.280,-179.695,19.618,152.217
C01400=1103.153,425.115,-98.239,-179.696,19.609,152.215
C01401=1103.147,424.894,-98.203,-179.698,19.601,152.213
C01402=1103.142,424.673,-98.167,-179.700,19.593,152.212
C01403=1103.138,424.451,-98.131,-179.701,19.586,152.210
C01404=1103.132,424.231,-98.095,-179.703,19.578,152.208
C01405=1103.127,424.010,-98.058,-179.705,19.570,152.207
C01406=1103.122,423.790,-98.023,-179.707,19.562,152.205
C01407=1103.116,423.569,-97.986,-179.708,19.554,152.203
C01408=1103.112,423.348,-97.950,-179.710,19.546,152.202
C01409=1103.106,423.101,-97.911,-179.712,19.538,152.200
C01410=1103.100,422.854,-97.870,-179.714,19.529,152.198
C01411=1103.094,422.608,-97.830,-179.716,19.521,152.196
C01412=1103.089,422.361,-97.790,-179.718,19.513,152.195
C01413=1103.083,422.114,-97.750,-179.720,19.504,152.193
C01414=1103.076,421.868,-97.710,-179.722,19.496,152.191
C01415=1103.072,421.621,-97.670,-179.724,19.487,152.189
C01416=1103.065,421.375,-97.630,-179.726,19.479,152.188
C01417=1103.060,421.128,-97.589,-179.727,19.471,152.186
C01418=1103.053,420.881,-97.550,-179.730,19.463,152.184
C01419=1103.048,420.635,-97.510,-179.732,19.454,152.182
C01420=1103.042,420.387,-97.470,-179.733,19.446,152.181
C01421=1103.036,420.141,-97.430,-179.736,19.438,152.179
C01422=1103.030,419.895,-97.390,-179.738,19.429,152.177
C01423=1103.025,419.648,-97.350,-179.740,19.421,152.176
C01424=1103.019,419.400,-97.310,-179.742,19.413,152.174
C01425=1103.013,419.155,-97.271,-179.744,19.405,152.172
C01426=1103.008,418.907,-97.231,-179.746,19.397,152.171
C01427=1103.001,418.661,-97.191,-179.748,19.389,152.169
C01428=1102.996,418.414,-97.151,-179.750,19.381,152.167
C01429=1102.990,418.167,-97.111,-179.752,19.373,152.166
C01430=1102.984,417.920,-97.071,-179.754,19.365,152.164
C01431=1102.979,417.674,-97.032,-179.756,19.357,152.162
C01432=1102.972,417.427,-96.992,-179.758,19.349,152.161
C01433=1102.968,417.181,-96.952,-179.761,19.341,152.159
C01434=1102.961,416.933,-96.913,-179.763,19.333,152.158
C01435=1102.955,416.686,-96.874,-179.764,19.326,152.156
C01436=1102.950,416.441,-96.834,-179.766,19.318,152.154
C01437=1102.944,416.193,-96.794,-179.769,19.310,152.153
C01438=1102.938,415.946,-96.754,-179.771,19.302,152.151
C01439=1102.933,415.700,-96.715,-179.773,19.294,152.150
C01440=1102.927,415.452,-96.676,-179.775,19.286,152.148
C01441=1102.921,415.207,-96.636,-179.777,19.279,152.147
C01442=1102.915,414.959,-96.597,-179.779,19.272,152.145
C01443=1102.909,414.712,-96.557,-179.782,19.264,152.144
C01444=1102.903,414.466,-96.518,-179.784,19.256,152.142
C01445=1102.897,414.219,-96.479,-179.786,19.249,152.141
C01446=1102.892,413.972,-96.440,-179.788,19.242,152.139
C01447=1102.886,413.725,-96.400,-179.790,19.234,152.138
C01448=1102.880,413.478,-96.361,-179.792,19.226,152.136
C01449=1102.874,413.232,-96.322,-179.795,19.219,152.135
C01450=1102.868,412.984,-96.282,-179.796,19.212,152.133
C01451=1102.863,412.738,-96.243,-179.799,19.204,152.132
C01452=1102.856,412.491,-96.204,-179.801,19.197,152.130
C01453=1102.851,412.244,-96.165,-179.804,19.189,152.129
C01454=1102.845,411.997,-96.125,-179.805,19.182,152.128
C01455=1102.839,411.751,-96.086,-179.808,19.175,152.126
C01456=1102.833,411.504,-96.047,-179.810,19.167,152.125
C01457=1102.828,411.289,-96.013,-179.812,19.161,152.124
C01458=1102.824,411.076,-95.979,-179.814,19.154,152.122
C01459=1102.819,410.862,-95.946,-179.815,19.149,152.121
C01460=1102.814,410.647,-95.911,-179.817,19.143,152.120
C01461=1102.809,410.433,-95.877,-179.819,19.136,152.119
C01462=1102.804,410.218,-95.843,-179.821,19.130,152.117
C01463=1102.799,410.005,-95.809,-179.823,19.124,152.116
C01464=1102.794,409.791,-95.776,-179.825,19.118,152.115
C01465=1102.788,409.544,-95.736,-179.827,19.110,152.114
C01466=1102.783,409.297,-95.698,-179.829,19.103,152.112
C01467=1102.777,409.050,-95.659,-179.832,19.096,152.111
C01468=1102.771,408.803,-95.620,-179.834,19.090,152.110
C01469=1102.765,408.556,-95.582,-179.836,19.082,152.108
C01470=1102.759,408.309,-95.542,-179.839,19.075,152.107
C01471=1102.754,408.063,-95.503,-179.840,19.069,152.106
C01472=1102.749,407.816,-95.465,-179.843,19.061,152.104
C01473=1102.743,407.569,-95.426,-179.845,19.055,152.103
C01474=1102.737,407.322,-95.388,-179.847,19.047,152.102
C01475=1102.731,407.075,-95.348,-179.849,19.041,152.100
C01476=1102.726,406.828,-95.310,-179.852,19.034,152.099
C01477=1102.720,406.581,-95.271,-179.854,19.027,152.098
C01478=1102.714,406.334,-95.233,-179.856,19.021,152.097
C01479=1102.708,406.087,-95.194,-179.858,19.014,152.095
C01480=1102.702,405.840,-95.155,-179.861,19.007,152.094
C01481=1102.697,405.593,-95.116,-179.863,19.000,152.093
C01482=1102.691,405.346,-95.078,-179.866,18.994,152.091
C01483=1102.685,405.099,-95.039,-179.868,18.987,152.090
C01484=1102.680,404.852,-95.000,-179.870,18.980,152.089
C01485=1102.674,404.605,-94.963,-179.872,18.974,152.088
C01486=1102.668,404.358,-94.923,-179.875,18.967,152.087
C01487=1102.662,404.112,-94.886,-179.877,18.961,152.085
C01488=1102.657,403.864,-94.847,-179.880,18.954,152.084
C01489=1102.651,403.617,-94.808,-179.882,18.948,152.083
C01490=1102.645,403.371,-94.770,-179.884,18.941,152.082
C01491=1102.639,403.124,-94.732,-179.886,18.935,152.081
C01492=1102.633,402.877,-94.693,-179.888,18.928,152.079
C01493=1102.628,402.630,-94.654,-179.891,18.922,152.078
C01494=1102.622,402.383,-94.617,-179.893,18.915,152.077
C01495=1102.616,402.135,-94.578,-179.895,18.909,152.076
C01496=1102.610,401.888,-94.540,-179.898,18.903,152.075
C01497=1102.604,401.642,-94.501,-179.900,18.896,152.074
C01498=1102.599,401.395,-94.463,-179.903,18.890,152.073
C01499=1102.593,401.147,-94.425,-179.905,18.884,152.071
C01500=1102.587,400.901,-94.387,-179.907,18.877,152.070
C01501=1102.582,400.654,-94.349,-179.910,18.871,152.069
C01502=1102.576,400.407,-94.311,-179.912,18.865,152.068
C01503=1102.571,400.160,-94.272,-179.914,18.859,152.067
C01504=1102.564,399.912,-94.234,-179.917,18.852,152.066
C01505=1102.559,399.665,-94.196,-179.919,18.846,152.065
C01506=1102.553,399.419,-94.158,-179.921,18.840,152.064
C01507=1102.547,399.172,-94.120,-179.924,18.834,152.063
C01508=1102.541,398.924,-94.082,-179.926,18.828,152.061
C01509=1102.535,398.677,-94.044,-179.929,18.822,152.060
C01510=1102.530,398.431,-94.006,-179.931,18.816,152.059
C01511=1102.524,398.184,-93.968,-179.934,18.809,152.058
C01512=1102.519,397.937,-93.930,-179.936,18.804,152.057
C01513=1102.513,397.723,-93.897,-179.938,18.799,152.056
C01514=1102.509,397.508,-93.865,-179.940,18.793,152.055
C01515=1102.503,397.294,-93.832,-179.943,18.788,152.055
C01516=1102.498,397.080,-93.798,-179.944,18.783,152.054
C01517=1102.493,396.866,-93.766,-179.947,18.778,152.053
C01518=1102.489,396.652,-93.733,-179.948,18.773,152.052
C01519=1102.483,396.438,-93.700,-179.951,18.767,152.051
C01520=1102.479,396.223,-93.667,-179.953,18.762,152.050
C01521=1102.473,395.976,-93.630,-179.955,18.757,152.049
C01522=1102.467,395.730,-93.592,-179.958,18.751,152.048
C01523=1102.461,395.483,-93.554,-179.960,18.745,152.047
C01524=1102.456,395.235,-93.516,-179.962,18.739,152.046
C01525=1102.450,394.989,-93.479,-179.965,18.733,152.045
C01526=1102.444,394.742,-93.441,-179.967,18.728,152.044
C01527=1102.438,394.494,-93.403,-179.970,18.721,152.043
C01528=1102.432,394.247,-93.366,-179.973,18.716,152.042
C01529=1102.426,394.000,-93.328,-179.975,18.710,152.041
C01530=1102.421,393.753,-93.291,-179.977,18.705,152.040
C01531=1102.416,393.506,-93.253,-179.980,18.699,152.039
C01532=1102.410,393.259,-93.215,-179.982,18.693,152.038
C01533=1102.404,393.012,-93.178,-179.985,18.687,152.038
C01534=1102.398,392.765,-93.140,-179.987,18.681,152.037
C01535=1102.392,392.518,-93.103,-179.990,18.676,152.036
C01536=1102.387,392.271,-93.065,-179.992,18.671,152.035
C01537=1102.381,392.024,-93.027,-179.995,18.665,152.034
C01538=1102.375,391.777,-92.990,-179.997,18.660,152.033
C01539=1102.369,391.530,-92.953,-180.000,18.654,152.032
C01540=1102.364,391.283,-92.916,179.998,18.649,152.031
C01541=1102.358,391.036,-92.878,179.995,18.643,152.030
C01542=1102.352,390.789,-92.841,179.992,18.637,152.029
C01543=1102.346,390.542,-92.803,179.989,18.632,152.029
C01544=1102.340,390.295,-92.767,179.987,18.627,152.028
C01545=1102.334,390.047,-92.730,179.985,18.621,152.027
C01546=1102.328,389.801,-92.692,179.982,18.616,152.026
C01547=1102.323,389.553,-92.655,179.979,18.611,152.025
C01548=1102.317,389.307,-92.617,179.977,18.605,152.024
C01549=1102.311,389.059,-92.580,179.975,18.600,152.023
C01550=1102.306,388.812,-92.543,179.972,18.595,152.023
C01551=1102.300,388.565,-92.505,179.969,18.589,152.022
C01552=1102.293,388.318,-92.469,179.966,18.584,152.021
C01553=1102.288,388.071,-92.432,179.964,18.578,152.020
C01554=1102.282,387.823,-92.395,179.961,18.573,152.019
C01555=1102.277,387.577,-92.357,179.958,18.568,152.018
C01556=1102.271,387.330,-92.320,179.956,18.563,152.018
C01557=1102.266,387.082,-92.283,179.953,18.557,152.017
C01558=1102.259,386.835,-92.247,179.951,18.552,152.016
C01559=1102.253,386.589,-92.209,179.948,18.547,152.015
C01560=1102.248,386.341,-92.172,179.946,18.541,152.014
C01561=1102.242,386.094,-92.135,179.943,18.536,152.014
C01562=1102.237,385.847,-92.098,179.940,18.531,152.013
C01563=1102.231,385.600,-92.062,179.937,18.526,152.012
C01564=1102.225,385.353,-92.025,179.935,18.521,152.011
C01565=1102.220,385.106,-91.988,179.932,18.516,152.011
C01566=1102.214,384.858,-91.951,179.930,18.511,152.010
C01567=1102.208,384.611,-91.914,179.927,18.506,152.009
C01568=1102.203,384.364,-91.878,179.924,18.501,152.008
C01569=1102.193,383.949,-91.815,179.920,18.492,152.007
C01570=1102.183,383.533,-91.753,179.915,18.483,152.006
C01571=1102.173,383.116,-91.692,179.911,18.475,152.005
C01572=1102.164,382.701,-91.630,179.907,18.467,152.003
C01573=1102.159,382.453,-91.593,179.904,18.462,152.003
C01574=1102.152,382.206,-91.557,179.901,18.457,152.002
C01575=1102.147,381.959,-91.520,179.898,18.452,152.001
C01576=1102.142,381.712,-91.483,179.896,18.447,152.001
C01577=1102.135,381.465,-91.446,179.893,18.443,152.000
C01578=1102.130,381.217,-91.410,179.890,18.437,151.999
C01579=1102.124,380.970,-91.374,179.887,18.432,151.999
C01580=1102.118,380.723,-91.337,179.885,18.428,151.998
C01581=1102.112,380.477,-91.301,179.882,18.423,151.997
C01582=1102.107,380.229,-91.263,179.879,18.418,151.997
C01583=1102.101,379.981,-91.228,179.876,18.413,151.996
C01584=1102.095,379.734,-91.191,179.874,18.409,151.995
C01585=1102.089,379.488,-91.155,179.871,18.404,151.995
C01586=1102.083,379.240,-91.119,179.869,18.399,151.994
C01587=1102.078,378.993,-91.082,179.866,18.394,151.993
C01588=1102.072,378.746,-91.046,179.863,18.390,151.993
C01589=1102.067,378.498,-91.009,179.860,18.385,151.992
C01590=1102.060,378.251,-90.973,179.857,18.380,151.991
C01591=1102.055,378.004,-90.936,179.854,18.375,151.991
C01592=1102.049,377.757,-90.901,179.852,18.371,151.990
C01593=1102.044,377.510,-90.864,179.849,18.367,151.990
C01594=1102.038,377.262,-90.828,179.846,18.362,151.989
C01595=1102.032,377.016,-90.792,179.844,18.357,151.988
C01596=1102.027,376.768,-90.755,179.841,18.352,151.988
C01597=1102.020,376.521,-90.719,179.838,18.348,151.987
C01598=1102.016,376.273,-90.683,179.836,18.343,151.986
C01599=1102.009,376.026,-90.647,179.833,18.339,151.986
C01600=1102.004,375.779,-90.611,179.830,18.334,151.985
C01601=1101.998,375.532,-90.574,179.827,18.329,151.985
C01602=1101.992,375.284,-90.538,179.824,18.325,151.984
C01603=1101.987,375.038,-90.502,179.821,18.320,151.984
C01604=1101.981,374.790,-90.466,179.819,18.316,151.983
C01605=1101.975,374.542,-90.430,179.816,18.311,151.982
C01606=1101.970,374.296,-90.394,179.813,18.307,151.982
C01607=1101.964,374.048,-90.358,179.810,18.302,151.981
C01608=1101.959,373.801,-90.323,179.807,18.298,151.981
C01609=1101.952,373.554,-90.286,179.805,18.294,151.980
C01610=1101.946,373.306,-90.250,179.802,18.289,151.980
C01611=1101.941,373.059,-90.215,179.799,18.285,151.979
C01612=1101.935,372.812,-90.179,179.796,18.281,151.979
C01613=1101.929,372.564,-90.142,179.793,18.276,151.978
C01614=1101.924,372.317,-90.107,179.790,18.272,151.978
C01615=1101.918,372.069,-90.071,179.787,18.267,151.977
C01616=1101.912,371.823,-90.035,179.784,18.263,151.977
C01617=1101.906,371.575,-89.999,179.782,18.259,151.976
C01618=1101.900,371.328,-89.964,179.779,18.255,151.976
C01619=1101.895,371.081,-89.928,179.776,18.250,151.975
C01620=1101.889,370.833,-89.893,179.773,18.246,151.975
C01621=1101.880,370.444,-89.836,179.769,18.240,151.974
C01622=1101.871,370.055,-89.779,179.765,18.233,151.973
C01623=1101.862,369.667,-89.724,179.760,18.226,151.972
C01624=1101.854,369.277,-89.668,179.755,18.220,151.971
C01625=1101.848,369.029,-89.632,179.752,18.215,151.971
C01626=1101.842,368.782,-89.597,179.749,18.211,151.971
C01627=1101.836,368.535,-89.561,179.747,18.207,151.970
C01628=1101.831,368.288,-89.526,179.744,18.203,151.970
C01629=1101.825,368.040,-89.490,179.741,18.199,151.969
C01630=1101.819,367.793,-89.455,179.738,18.195,151.969
C01631=1101.813,367.545,-89.419,179.735,18.191,151.968
C01632=1101.808,367.298,-89.384,179.732,18.186,151.968
C01633=1101.802,367.051,-89.348,179.729,18.182,151.967
C01634=1101.796,366.804,-89.312,179.726,18.178,151.967
C01635=1101.791,366.557,-89.277,179.723,18.174,151.966
C01636=1101.785,366.308,-89.242,179.720,18.170,151.966
C01637=1101.780,366.062,-89.207,179.718,18.166,151.966
C01638=1101.774,365.814,-89.171,179.714,18.162,151.965
C01639=1101.768,365.567,-89.136,179.711,18.158,151.965
C01640=1101.762,365.319,-89.100,179.709,18.154,151.964
C01641=1101.757,365.072,-89.065,179.706,18.150,151.964
C01642=1101.750,364.824,-89.030,179.703,18.146,151.964
C01643=1101.745,364.577,-88.995,179.700,18.142,151.963
C01644=1101.739,364.330,-88.959,179.697,18.138,151.963
C01645=1101.734,364.082,-88.924,179.694,18.134,151.962
C01646=1101.728,363.835,-88.889,179.691,18.130,151.962
C01647=1101.722,363.588,-88.854,179.688,18.126,151.961
C01648=1101.716,363.340,-88.819,179.685,18.122,151.961
C01649=1101.710,363.092,-88.784,179.682,18.119,151.961
C01650=1101.705,362.845,-88.749,179.680,18.115,151.960
C01651=1101.700,362.598,-88.714,179.676,18.111,151.960
C01652=1101.693,362.350,-88.678,179.673,18.107,151.960
C01653=1101.688,362.103,-88.644,179.670,18.103,151.959
C01654=1101.682,361.855,-88.608,179.667,18.099,151.959
C01655=1101.677,361.608,-88.573,179.665,18.096,151.959
C01656=1101.671,361.361,-88.539,179.661,18.092,151.958
C01657=1101.665,361.113,-88.504,179.658,18.088,151.958
C01658=1101.659,360.866,-88.468,179.656,18.084,151.957
C01659=1101.654,360.618,-88.434,179.652,18.080,151.957
C01660=1101.648,360.371,-88.398,179.650,18.077,151.957
C01661=1101.642,360.123,-88.364,179.646,18.073,151.956
C01662=1101.636,359.875,-88.328,179.643,18.069,151.956
C01663=1101.631,359.628,-88.294,179.641,18.065,151.956
C01664=1101.625,359.381,-88.259,179.637,18.061,151.955
C01665=1101.619,359.133,-88.224,179.635,18.058,151.955
C01666=1101.614,358.886,-88.190,179.631,18.054,151.955
C01667=1101.608,358.638,-88.155,179.628,18.051,151.955
C01668=1101.602,358.391,-88.120,179.625,18.047,151.954
C01669=1101.597,358.143,-88.085,179.623,18.043,151.954
C01670=1101.591,357.896,-88.051,179.619,18.040,151.954
C01671=1101.585,357.648,-88.015,179.617,18.036,151.953
C01672=1101.579,357.401,-87.981,179.613,18.032,151.953
C01673=1101.570,357.026,-87.929,179.608,18.027,151.953
C01674=1101.562,356.653,-87.876,179.604,18.021,151.952
C01675=1101.553,356.278,-87.824,179.599,18.015,151.952
C01676=1101.545,355.904,-87.772,179.595,18.011,151.951
C01677=1101.539,355.656,-87.738,179.592,18.007,151.951
C01678=1101.533,355.409,-87.702,179.589,18.003,151.951
C01679=1101.527,355.162,-87.668,179.586,18.000,151.950
C01680=1101.522,354.915,-87.634,179.583,17.997,151.950
C01681=1101.516,354.667,-87.599,179.580,17.993,151.950
C01682=1101.511,354.419,-87.565,179.577,17.990,151.950
C01683=1101.505,354.172,-87.531,179.573,17.986,151.949
C01684=1101.500,353.924,-87.496,179.571,17.982,151.949
C01685=1101.494,353.677,-87.462,179.567,17.979,151.949
C01686=1101.488,353.428,-87.427,179.565,17.975,151.948
C01687=1101.482,353.181,-87.393,179.561,17.972,151.948
C01688=1101.476,352.934,-87.359,179.558,17.969,151.948
C01689=1101.471,352.686,-87.324,179.555,17.965,151.948
C01690=1101.465,352.438,-87.290,179.552,17.962,151.948
C01691=1101.459,352.191,-87.256,179.549,17.958,151.947
C01692=1101.454,351.943,-87.221,179.546,17.955,151.947
C01693=1101.448,351.696,-87.187,179.542,17.951,151.947
C01694=1101.442,351.449,-87.153,179.540,17.948,151.947
C01695=1101.437,351.200,-87.119,179.537,17.945,151.946
C01696=1101.431,350.953,-87.084,179.533,17.941,151.946
C01697=1101.425,350.705,-87.050,179.531,17.938,151.946
C01698=1101.419,350.458,-87.016,179.527,17.935,151.946
C01699=1101.414,350.211,-86.982,179.525,17.931,151.946
C01700=1101.408,349.963,-86.948,179.521,17.928,151.945
C01701=1101.402,349.715,-86.914,179.518,17.925,151.945
C01702=1101.396,349.467,-86.880,179.515,17.922,151.945
C01703=1101.391,349.220,-86.845,179.512,17.918,151.945
C01704=1101.385,348.972,-86.811,179.509,17.915,151.945
C01705=1101.379,348.725,-86.778,179.506,17.911,151.944
C01706=1101.374,348.477,-86.744,179.503,17.908,151.944
C01707=1101.368,348.230,-86.709,179.499,17.905,151.944
C01708=1101.363,347.982,-86.676,179.496,17.902,151.944
C01709=1101.356,347.734,-86.641,179.493,17.899,151.944
C01710=1101.351,347.487,-86.607,179.490,17.895,151.943
C01711=1101.345,347.239,-86.574,179.487,17.892,151.943
C01712=1101.339,346.991,-86.540,179.483,17.888,151.943
C01713=1101.334,346.743,-86.506,179.481,17.886,151.943
C01714=1101.329,346.496,-86.472,179.478,17.882,151.943
C01715=1101.323,346.249,-86.438,179.474,17.879,151.943
C01716=1101.317,346.001,-86.405,179.471,17.876,151.942
C01717=1101.311,345.753,-86.371,179.469,17.873,151.942
C01718=1101.306,345.505,-86.337,179.465,17.869,151.942
C01719=1101.300,345.258,-86.303,179.462,17.866,151.942
C01720=1101.294,345.010,-86.270,179.459,17.863,151.942
C01721=1101.288,344.763,-86.236,179.456,17.860,151.942
C01722=1101.283,344.515,-86.202,179.453,17.857,151.942
C01723=1101.277,344.266,-86.169,179.449,17.854,151.941
C01724=1101.271,344.019,-86.135,179.446,17.851,151.941
C01725=1101.263,343.647,-86.085,179.442,17.846,151.941
C01726=1101.254,343.276,-86.034,179.437,17.842,151.941
C01727=1101.246,342.904,-85.984,179.432,17.837,151.941
C01728=1101.237,342.531,-85.933,179.427,17.833,151.941
C01729=1101.231,342.284,-85.900,179.424,17.830,151.940
C01730=1101.225,342.036,-85.866,179.421,17.826,151.940
C01731=1101.220,341.789,-85.833,179.418,17.823,151.940
C01732=1101.214,341.541,-85.799,179.415,17.821,151.940
C01733=1101.208,341.293,-85.765,179.411,17.817,151.940
C01734=1101.203,341.045,-85.732,179.408,17.814,151.940
C01735=1101.197,340.798,-85.699,179.405,17.811,151.940
C01736=1101.191,340.550,-85.665,179.402,17.808,151.940
C01737=1101.186,340.302,-85.631,179.399,17.806,151.940
C01738=1101.181,340.055,-85.598,179.396,17.803,151.939
C01739=1101.174,339.808,-85.566,179.393,17.800,151.939
C01740=1101.169,339.560,-85.532,179.389,17.796,151.939
C01741=1101.163,339.312,-85.499,179.386,17.794,151.939
C01742=1101.158,339.064,-85.466,179.383,17.791,151.939
C01743=1101.152,338.817,-85.432,179.379,17.788,151.939
C01744=1101.146,338.569,-85.398,179.376,17.785,151.939
C01745=1101.140,338.321,-85.366,179.374,17.782,151.939
C01746=1101.135,338.073,-85.332,179.370,17.779,151.939
C01747=1101.129,337.825,-85.299,179.367,17.776,151.939
C01748=1101.123,337.577,-85.266,179.364,17.773,151.939
C01749=1101.117,337.330,-85.233,179.361,17.771,151.939
C01750=1101.112,337.082,-85.199,179.358,17.768,151.938
C01751=1101.106,336.834,-85.166,179.354,17.765,151.938
C01752=1101.100,336.587,-85.134,179.351,17.762,151.938
C01753=1101.095,336.339,-85.100,179.348,17.760,151.938
C01754=1101.089,336.091,-85.067,179.345,17.757,151.938
C01755=1101.084,335.843,-85.034,179.341,17.753,151.938
C01756=1101.077,335.596,-85.001,179.338,17.751,151.938
C01757=1101.072,335.347,-84.968,179.335,17.748,151.938
C01758=1101.066,335.100,-84.936,179.332,17.745,151.938
C01759=1101.060,334.852,-84.902,179.328,17.742,151.938
C01760=1101.055,334.605,-84.869,179.325,17.740,151.938
C01761=1101.049,334.357,-84.837,179.322,17.737,151.938
C01762=1101.043,334.109,-84.803,179.319,17.734,151.938
C01763=1101.038,333.861,-84.770,179.315,17.731,151.938
C01764=1101.032,333.613,-84.738,179.312,17.728,151.938
C01765=1101.027,333.366,-84.705,179.309,17.726,151.938
C01766=1101.021,333.118,-84.672,179.306,17.723,151.938
C01767=1101.015,332.870,-84.639,179.303,17.721,151.938
C01768=1101.010,332.622,-84.606,179.299,17.717,151.938
C01769=1101.004,332.374,-84.573,179.296,17.715,151.938
C01770=1100.999,332.127,-84.540,179.293,17.712,151.938
C01771=1100.993,331.879,-84.508,179.290,17.710,151.938
C01772=1100.987,331.631,-84.475,179.287,17.707,151.938
C01773=1100.981,331.383,-84.442,179.284,17.705,151.938
C01774=1100.975,331.135,-84.410,179.280,17.702,151.938
C01775=1100.969,330.887,-84.377,179.277,17.699,151.938
C01776=1100.964,330.640,-84.345,179.274,17.697,151.938
C01777=1100.955,330.262,-84.294,179.269,17.693,151.938
C01778=1100.946,329.884,-84.245,179.263,17.689,151.938
C01779=1100.937,329.506,-84.196,179.259,17.685,151.938
C01780=1100.929,329.128,-84.146,179.254,17.681,151.938
C01781=1100.923,328.880,-84.113,179.251,17.679,151.938
C01782=1100.917,328.632,-84.081,179.247,17.676,151.938
C01783=1100.911,328.384,-84.048,179.244,17.673,151.938
C01784=1100.906,328.137,-84.016,179.241,17.671,151.938
C01785=1100.899,327.889,-83.983,179.237,17.668,151.938
C01786=1100.893,327.641,-83.951,179.234,17.666,151.938
C01787=1100.888,327.392,-83.919,179.231,17.663,151.938
C01788=1100.882,327.146,-83.886,179.228,17.661,151.938
C01789=1100.876,326.897,-83.854,179.224,17.658,151.938
C01790=1100.871,326.649,-83.821,179.221,17.655,151.938
C01791=1100.865,326.402,-83.789,179.218,17.653,151.938
C01792=1100.859,326.154,-83.757,179.215,17.651,151.938
C01793=1100.853,325.906,-83.725,179.211,17.648,151.938
C01794=1100.848,325.658,-83.692,179.208,17.646,151.938
C01795=1100.843,325.410,-83.660,179.205,17.643,151.938
C01796=1100.836,325.162,-83.627,179.202,17.641,151.938
C01797=1100.831,324.915,-83.596,179.198,17.639,151.939
C01798=1100.825,324.667,-83.564,179.194,17.636,151.939
